VAR_INPUT
	{attribute 'OPC.UA.DA' := '1'}
	rAlarmHigh : REAL;
	{attribute 'OPC.UA.DA' := '1'}
	rAlarmLow : REAL;
	{attribute 'OPC.UA.DA' := '1'}
	rLimitHigh : REAL; // the upper limit of the desirable range (when the downward adjustment is activated)
	{attribute 'OPC.UA.DA' := '1'}
	rLimitLow : REAL; // lower limit of the desirable range (when the upward adjustment is activated)
	{attribute 'OPC.UA.DA' := '1'}
	nAdjustDelay : REAL; // min time in seconds between adjustments
	{attribute 'OPC.UA.DA' := '1'}
	nProcessValue : REAL; 
	{attribute 'OPC.UA.DA' := '1'}
	bEnabled : BOOL; 
	{attribute 'OPC.UA.DA' := '1'}
	rCurrentValue : REAL; 
	{attribute 'OPC.UA.DA' := '1'}
	sParameterName : STRING;
	{attribute 'OPC.UA.DA' := '1'}
	rSetpoint: REAL;
	{attribute 'OPC.UA.DA' := '1'}
	Mode:    E_CTRL_MODE;
END_VAR


VAR PERSISTENT

	n_ProcessValue: FLOAT;
	
	{attribute 'OPC.UA.DA' := '1'} 
	tPIDLoopTime: TIME := T#1M;	// how often the PID loop should be executed
	tResetMister: TIME := T#20M;	// reset the humidifiers every 20m so that the output doesn't get stuck high with mister ON timer expired causing mister to turn off
	
	// PID loop variables below
	nPID_Setpoint:			REAL; 
	nPID_SetpointBand:		REAL; // 
	nPID_ManSyncVal:		REAL;
	bPID_Sync: 				BOOL;
	nPID_Error:				REAL;
	nPID_ErrorPerc:			REAL;  
	nPID_Output: 			LREAL; 
	bPID_Hold: 				BOOL;
	ePID_Mode: 				E_CTRL_MODE;
	stPID_Parameters: 		ST_CTRL_PID_PARAMS;
	ePID_ErrorId: 			E_CTRL_ERRORCODES;
	bPID_Error: 			BOOL;
	bPID_ARWactive: 		BOOL;
	
	//stPIDParams values
	tPID_CtrlCycleTime: 		TIME := tPIDLoopTime;
	tPID_TaskCycleTime:			TIME := T#10MS;
	nPID_Kp:  					REAL := 1.0;
	nPID_Compensator:  			REAL := 1.0/1000.0;
	tPID_Tn: 					TIME := T#0S;
	tPID_Tv:					TIME := T#0S;
	tPID_Td:					TIME := T#200S; 
	nPID_OutMaxLimit: 			REAL := 300; 		// this is set in the cyclic routine, the error band moves with the setpoint
	nPID_OutMinLimit:			REAL := 0;
	bPID_PInTheFeedbackPath: 	BOOL := FALSE;
	bPID_DInTheFeedbackPath: 	BOOL := FALSE;
	bPID_ARWOnIPartOnly:		BOOL := FALSE;
	
	n_Output: LREAL := 0;
	
END_VAR

VAR
	bFirstRun: BOOL := TRUE;
	bResetTimer: BOOL := FALSE;
	
	eSMState: 	(WAIT, CALCULATE, TRIG_UP, TRIG_DOWN) := WAIT;

	{attribute 'OPC.UA.DA' := '0'} 
	fbTON_PIDLoop: TON := (PT := tPIDLoopTime, IN := FALSE);
	
	fbTON_OPCUATagReset: TON := (PT := T#1S, IN := FALSE);
	
	fbTON_ResetMister: TON := (PT := tResetMister, IN := FALSE);
	fbTON_ResetMisterCountdown: TON := (PT := T#1S, IN := FALSE);
	
	{attribute 'OPC.UA.DA' := '0'}
	PID: FB_CTRL_PID;
	
END_VAR


VAR_OUTPUT
	{attribute 'OPC.UA.DA' := '1'}
	bAdjustDownOutput 		AT %Q*: BOOL;
	{attribute 'OPC.UA.DA' := '1'}
	bAdjustUpOutput 		AT %Q*: BOOL;
	{attribute 'OPC.UA.DA' := '1'}
	bAlarmHigh : 			BOOL;
	{attribute 'OPC.UA.DA' := '1'}
	bAlarmLow : 			BOOL;
END_VAR


VAR
	fbTON_AdjustDown : 		TON;
	fbTON_AdjustUp : 		TON;
	{attribute 'OPC.UA.DA' := '1'}
	tAdjustUp : 			TIME;
	tAdjustDown : 			TIME;
	tAdjustUpCTRL : 			TIME; // these variables created to enable continuous misting - Ignition requires tAdjustUp/Down to be reset to 0 after each dose to enable plotting
	tAdjustDownCTRL : 			TIME;
	
END_VAR

IF bFirstRun THEN
	fbTON_PIDLoop(PT := tPIDLoopTime, IN := TRUE);
	fbTON_ResetMister(PT := tResetMister, IN := TRUE);
	bFirstRun := FALSE;
END_IF

//eState := eStateTarget;

IF (NOT bEnable) OR (eState = E_DeviceState.IDLE) THEN
	eState := E_DeviceState.IDLE;
	eStateTarget := E_DeviceState.IDLE;
	PID.eMode := E_CTRL_MODE.eCTRL_MODE_RESET;
END_IF

IF bEnable AND (eState = E_DeviceState.RUNNING) THEN
	PID.eMode := E_CTRL_MODE.eCTRL_MODE_ACTIVE;
END_IF 



// Execute timers
fbTON_PIDLoop(PT := tPIDLoopTime);
fbTON_OPCUATagReset();
fbTON_ResetMister();
fbTON_ResetMisterCountdown();

fbTON_AdjustUp();
fbTON_AdjustDown();

updatePIDParams();

nPID_Error 	:= nPID_Setpoint - nProcessValue; // calcuate error

nPID_Setpoint := (rLimitHigh + rLimitLow) / 2.0;
rSetpoint := (rLimitHigh + rLimitLow) / 2.0;

// nPID_Setpoint := 67;

rCurrentValue := nProcessValue;

IF fbTON_AdjustUp.Q THEN
	bAdjustUpOutput := FALSE;
	fbTON_AdjustUp.IN := FALSE;
END_IF

(*
IF fbTON_AdjustDown.Q THEN
	bAdjustDownOutput := FALSE;          // DEHUMIDIFER STAYS ON
	fbTON_AdjustDown.IN := FALSE;
END_IF
*)
bAdjustDownOutput := TRUE; // this code was added to keep the dehumidifier always on - remove this when we start controlling the fan

IF eState = E_DeviceState.RUNNING THEN
	//PID.eMode := E_CTRL_MODE.eCTRL_MODE_ACTIVE;
	PID( fSetpointValue := nPID_Setpoint, fActualValue := nProcessValue, stParams := stPID_Parameters);
END_IF


// IF control loop is ON and the loop timer has elapsed then enter the calculate / action state machine below
IF fbTON_PIDLoop.Q AND (eState = E_DeviceState.RUNNING) THEN
	fbTON_PIDLoop.IN := FALSE;
	eSMState := CALCULATE;		// This is the entry point to start PID calculations and dosing
END_IF

IF fbTON_OPCUATagReset.Q AND (eState = E_DeviceState.RUNNING) THEN
	tAdjustDown := T#0MS;
	tAdjustUp := T#0MS;
	fbTON_OPCUATagReset.IN := FALSE;
END_IF


CASE eSMState OF

	WAIT:
		// Do nothing and wait for timer to trigger
		fbTON_PIDLoop(IN := TRUE);
		
	
	CALCULATE:
	
		IF (eState = E_DeviceState.RUNNING) THEN 
			IF PID.fOut > 0 AND NOT fbTON_ResetMister.Q THEN
				tAdjustUp 	:= REAL_TO_TIME(PID.fOut) * 1000;
				tAdjustUpCTRL 	:= REAL_TO_TIME(PID.fOut) * 1000;
				tAdjustDown := T#0MS;
				eSMState 	:= TRIG_UP;
			ELSIF PID.fOut < 0 THEN
				tAdjustDown	:= REAL_TO_TIME(-PID.fOut) *1000;
				tAdjustDownCTRL	:= REAL_TO_TIME(-PID.fOut) *1000;
				tAdjustUp := T#0MS;
				eSMState 	:= TRIG_DOWN;
			END_IF
		END_IF
			
		fbTON_PIDLoop(IN := FALSE);
		fbTON_OPCUATagReset(IN := TRUE);  // set the OPCUA tag reset timer (Ignition requires these tags to be set to 0 to be visible on graph)
		
		//eSMState := WAIT;
		IF (eSMState <> TRIG_UP) AND (eSMState <> TRIG_DOWN) THEN
			eSMState := WAIT;
		END_IF
		
		
	TRIG_UP:
		fbTON_AdjustUp(PT := tAdjustUpCTRL, IN := TRUE);  // start the timer for the duration set at PID output
		bAdjustUpOutput := TRUE; // set output to high
		eSMState := WAIT; // go back to wait for the next timer trigger
		fbTON_PIDLoop(IN := TRUE);	// restart the PID loop timer

		
		
	TRIG_DOWN:
		fbTON_AdjustDown(PT := tAdjustDownCTRL, IN := TRUE); // start the timer for the duration set at PID output
		bAdjustDownOutput := TRUE; // set output to high
		eSMState := WAIT; // go back to wait for the next timer trigger
		fbTON_PIDLoop(IN := TRUE);			
		
		
END_CASE

IF fbTON_ResetMister.Q THEN

	fbTON_ResetMisterCountdown(IN := TRUE);
	fbTON_ResetMister(IN := FALSE);
END_IF

IF fbTON_ResetMisterCountdown.IN THEN
		bAdjustUpOutput := FALSE;	
END_IF
IF fbTON_ResetMisterCountdown.Q THEN
		fbTON_ResetMisterCountdown(IN := FALSE);
		fbTON_ResetMister(IN := TRUE);
END_IF

METHOD FB_init : BOOL
VAR_INPUT
	bInitRetains : BOOL; // if TRUE, the retain variables are initialized (warm start / cold start)
	bInCopyCode : BOOL;  // if TRUE, the instance afterwards gets moved into the copy code (online change)
	

	
END_VAR
END_METHOD

METHOD setParams : BOOL
VAR_INPUT
	(*
	NutrientMaxDoseRate: UINT;
	NutrientMinDoseRate: UINT;
	NutrientTimeBetweenDoses: TIME;
	PHMaxDoseRate: UINT;
	PHMinDoseRate: UINT;
	PHTimeBetweenDoses: TIME;


	// PID loop variables below
	*)
	Setpoint:		REAL; 
	(*
	NutrientSetpointBand:	REAL;
	NutrientManSyncVal:		REAL;
	NutrientSync: 			BOOL; 
	NutrientHold: 			BOOL;
	NutrientMode: 			E_CTRL_MODE;
	NutrientCtrlCycleTime: 	TIME;
	NutrientTaskCycleTime:	TIME;
	
	//stPIDParams values
	NutrientKp:  				REAL;
	NutrientTn: 				TIME; 
	NutrientTv:					TIME; 
	NutrientTd:					TIME; 
	NutrientOutMaxLimit: 		REAL;
	NutrientOutMinLimit:		REAL;
	NutrientPInTheFeedbackPath: BOOL;
	NutrientDInTheFeedbackPath: BOOL;
	NutrientARWOnIPartOnly:		BOOL;
	
	*)
	PHSetpoint:			REAL; 
	(*
	PHSetpointBand:		REAL;
	PHManSyncVal:		REAL;
	PHSync: 			BOOL;
	PHHold: 			BOOL;
	PHMode: 			E_CTRL_MODE;
	PHCtrlCycleTime: 		TIME;
	PHTaskCycleTime:		TIME;
	
	
	//stPIDParams values
	PHKp:  					REAL;
	PHTn: 					TIME;
	PHTv:					TIME;
	PHTd:					TIME; 
	PHOutMaxLimit: 			REAL; 		
	PHOutMinLimit:			REAL;
	PHPInTheFeedbackPath: 	BOOL;
	PHDInTheFeedbackPath:	BOOL;
	PHARWOnIPartOnly:		BOOL;
	*)
	
END_VAR
(*
nPIDNutrientMaxDoseRate := 				NutrientMaxDoseRate;
nPIDNutrientMinDoseRate := 				NutrientMinDoseRate;
tPIDNutrientTimeBetweenDoses := 		NutrientTimeBetweenDoses;

nPIDPHMaxDoseRate := 					PHMaxDoseRate;
nPIDPHMinDoseRate := 					PHMinDoseRate;
tPIDPHTimeBetweenDoses := 				PHTimeBetweenDoses;

*)
nPID_Setpoint := 						Setpoint;
(*
nPIDNutrientSetpointBand := 			NutrientSetpointBand;
nPIDNutrientManSyncVal := 				NutrientManSyncVal;
bPIDNutrientSync := 					NutrientSync;
bPIDNutrientHold := 					NutrientHold;
ePIDNutrientMode := 					NutrientMode;
tPIDNutrientCtrlCycleTime := 			NutrientCtrlCycleTime;
tPIDNutrientTaskCycleTime := 			NutrientTaskCycleTime;

nPIDNutrientKp := 						NutrientKp;
tPIDNutrientTn := 						NutrientTn;
tPIDNutrientTv := 						NutrientTv;
tPIDNutrientTd := 						NutrientTd;
nPIDNutrientOutMaxLimit := 				NutrientOutMaxLimit;
nPIDNutrientOutMinLimit := 				NutrientOutMinLimit;
bPIDNutrientPInTheFeedbackPath := 		NutrientPInTheFeedbackPath;
bPIDNutrientDInTheFeedbackPath := 		NutrientDInTheFeedbackPath;
bPIDNutrientARWactive := 				NutrientARWOnIPartOnly;
*)
END_METHOD

METHOD setState : BOOL
VAR_INPUT
	state : E_DeviceState;
END_VAR

eState := state;
END_METHOD

METHOD updatePIDParams : BOOL
VAR_INPUT
END_VAR


stPID_Parameters.tCtrlCycleTime := 		tPID_CtrlCycleTime;
stPID_Parameters.tTaskCycleTime := 		tPID_TaskCycleTime;
stPID_Parameters.fKp := 				nPID_Kp;
stPID_Parameters.tTn := 				tPID_Tn;
stPID_Parameters.tTv := 				tPID_Tv;
stPID_Parameters.tTd := 				tPID_Td;
stPID_Parameters.fOutMaxLimit := 		nPID_OutMaxLimit;
stPID_Parameters.fOutMinLimit := 		nPID_OutMinLimit;
stPID_Parameters.bPInTheFeedbackPath := bPID_PInTheFeedbackPath;
stPID_Parameters.bDInTheFeedbackPath := bPID_DInTheFeedbackPath;
stPID_Parameters.bARWOnIPartOnly := 	bPID_ARWOnIPartOnly;
END_METHOD

END_FUNCTION_BLOCK

// ---- POUs/04 Control Loops/Dosing Machine/FB_ControlLoop_PID_HVAC.TcPOU
FUNCTION_BLOCK FB_ControlLoop_PID_HVAC EXTENDS FB_BaseDevice


VAR_INPUT
	{attribute 'OPC.UA.DA' := '1'}
	rAlarmHigh : REAL;
	{attribute 'OPC.UA.DA' := '1'}
	rAlarmLow : REAL;
	{attribute 'OPC.UA.DA' := '1'}
	rLimitHigh : REAL; // the upper limit of the desirable range (when the downward adjustment is activated)
	{attribute 'OPC.UA.DA' := '1'}
	rLimitLow : REAL; // lower limit of the desirable range (when the upward adjustment is activated)
	{attribute 'OPC.UA.DA' := '1'}
	nAdjustDelay : REAL; // min time in seconds between adjustments
	{attribute 'OPC.UA.DA' := '1'}
	nProcessValue : REAL; 
	{attribute 'OPC.UA.DA' := '1'}
	bEnabled : BOOL; 
	{attribute 'OPC.UA.DA' := '1'}
	rCurrentValue : REAL; 
	{attribute 'OPC.UA.DA' := '1'}
	sParameterName : STRING;
	{attribute 'OPC.UA.DA' := '1'}
	rSetpoint: REAL;
	{attribute 'OPC.UA.DA' := '1'}
	Mode:    E_CTRL_MODE;
END_VAR


VAR PERSISTENT

	n_ProcessValue: FLOAT;
	
	{attribute 'OPC.UA.DA' := '1'} 
	tPIDLoopTime: TIME := T#1M;	// how often the PID loop should be executed
	
	// PID loop variables below
	nPID_Setpoint:			REAL; 
	nPID_SetpointBand:		REAL; // 
	nPID_ManSyncVal:		REAL;
	bPID_Sync: 				BOOL;
	nPID_Error:				REAL;
	nPID_ErrorPerc:			REAL;  
	nPID_Output: 			LREAL; 
	bPID_Hold: 				BOOL;
	ePID_Mode: 				E_CTRL_MODE;
	stPID_Parameters: 		ST_CTRL_PID_PARAMS;
	ePID_ErrorId: 			E_CTRL_ERRORCODES;
	bPID_Error: 			BOOL;
	bPID_ARWactive: 		BOOL;
	
	//stPIDParams values
	tPID_CtrlCycleTime: 		TIME := tPIDLoopTime;
	tPID_TaskCycleTime:			TIME := T#10MS;
	nPID_Kp:  					REAL := 1.0;
	nPID_Compensator:  			REAL := 1.0/1000.0;
	tPID_Tn: 					TIME := T#0S;
	tPID_Tv:					TIME := T#0S;
	tPID_Td:					TIME := T#200S; 
	nPID_OutMaxLimit: 			REAL := 300; 		// this is set in the cyclic routine, the error band moves with the setpoint
	nPID_OutMinLimit:			REAL := 0;
	bPID_PInTheFeedbackPath: 	BOOL := FALSE;
	bPID_DInTheFeedbackPath: 	BOOL := FALSE;
	bPID_ARWOnIPartOnly:		BOOL := FALSE;
	
	n_Output: LREAL := 0;
	
END_VAR

VAR
	bFirstRun: BOOL := TRUE;
	bResetTimer: BOOL := FALSE;
	
	eSMState: 	(WAIT, CALCULATE, TRIG_UP, TRIG_DOWN) := WAIT;

	{attribute 'OPC.UA.DA' := '0'} 
	fbTON_PIDLoop: TON := (PT := tPIDLoopTime, IN := FALSE);
	
	{attribute 'OPC.UA.DA' := '0'}
	PID: FB_CTRL_PID;
	
END_VAR


VAR_OUTPUT
	{attribute 'OPC.UA.DA' := '1'}
	bAdjustDownOutput 		AT %Q*: BOOL;
	{attribute 'OPC.UA.DA' := '1'}
	bAdjustUpOutput 		AT %Q*: BOOL;
	{attribute 'OPC.UA.DA' := '1'}
	bAlarmHigh : 			BOOL;
	{attribute 'OPC.UA.DA' := '1'}
	bAlarmLow : 			BOOL;
	{attribute 'OPC.UA.DA' := '1'}
	nControlValue:			REAL;
END_VAR


VAR
	fbTON_AdjustDown : 		TON;
	fbTON_AdjustUp : 		TON;
	tAdjustUp : 			TIME;
	tAdjustDown : 			TIME;
	
	{attribute 'OPC.UA.DA' := '1'}
	nControlValue: POINTER TO REAL;
	{attribute 'OPC.UA.DA' := '1'}
	nControlValueCopy: REAL;
	
END_VAR

IF bFirstRun THEN
	fbTON_PIDLoop(PT := tPIDLoopTime, IN := TRUE);
	bFirstRun := FALSE;
END_IF

//eState := eStateTarget;

IF (NOT bEnable) OR (eState = E_DeviceState.IDLE) THEN
	eState := E_DeviceState.IDLE;
	eStateTarget := E_DeviceState.IDLE;
	PID.eMode := E_CTRL_MODE.eCTRL_MODE_RESET;
END_IF

IF bEnable AND (eState = E_DeviceState.RUNNING) THEN
	PID.eMode := E_CTRL_MODE.eCTRL_MODE_ACTIVE;
END_IF 



// Execute timers
fbTON_PIDLoop(PT := tPIDLoopTime);
fbTON_AdjustUp();
fbTON_AdjustDown();

updatePIDParams();

nPID_Error 	:= nPID_Setpoint - nProcessValue; // calcuate error

nPID_Setpoint := (rLimitHigh + rLimitLow) / 2.0;

// nPID_Setpoint := 67;

rCurrentValue := nProcessValue;

(*
IF fbTON_AdjustDown.Q THEN
	bAdjustDownOutput := FALSE;
	fbTON_AdjustDown.IN := FALSE;
END_IF
*)

IF eState = E_DeviceState.RUNNING THEN
	PID( fSetpointValue := nPID_Setpoint, fActualValue := nProcessValue, stParams := stPID_Parameters);
END_IF


// IF control loop is ON and the loop timer has elapsed then enter the calculate / action state machine below
IF fbTON_PIDLoop.Q AND (eState = E_DeviceState.RUNNING) THEN
	fbTON_PIDLoop.IN := FALSE;
	eSMState := CALCULATE;		// This is the entry point to start PID calculations and dosing
END_IF



CASE eSMState OF

	WAIT:
		// Do nothing and wait for timer to trigger
		fbTON_PIDLoop(IN := TRUE);
	
	CALCULATE:
	
		nControlValue := nControlValue + PID.fOut;
		fbTON_PIDLoop(IN := FALSE);
		
		eSMState := WAIT;
		

		
	TRIG_UP:
		fbTON_AdjustUp(PT := tAdjustUp, IN := TRUE);  // start the timer for the duration set at PID output
		bAdjustUpOutput := TRUE; // set output to high
		eSMState := WAIT; // go back to wait for the next timer trigger
		fbTON_PIDLoop(IN := TRUE);	// restart the PID loop timer

		
		
	TRIG_DOWN:
		fbTON_AdjustDown(PT := tAdjustDown, IN := TRUE); // start the timer for the duration set at PID output
		bAdjustDownOutput := TRUE; // set output to high
		eSMState := WAIT; // go back to wait for the next timer trigger
		fbTON_PIDLoop(IN := TRUE);			
		
		
END_CASE

METHOD FB_init : BOOL
VAR_INPUT
	bInitRetains : BOOL; // if TRUE, the retain variables are initialized (warm start / cold start)
	bInCopyCode : BOOL;  // if TRUE, the instance afterwards gets moved into the copy code (online change)
	

	
END_VAR
END_METHOD

METHOD setParams : BOOL
VAR_INPUT
	(*
	NutrientMaxDoseRate: UINT;
	NutrientMinDoseRate: UINT;
	NutrientTimeBetweenDoses: TIME;
	PHMaxDoseRate: UINT;
	PHMinDoseRate: UINT;
	PHTimeBetweenDoses: TIME;


	// PID loop variables below
	*)
	Setpoint:		REAL; 
	(*
	NutrientSetpointBand:	REAL;
	NutrientManSyncVal:		REAL;
	NutrientSync: 			BOOL; 
	NutrientHold: 			BOOL;
	NutrientMode: 			E_CTRL_MODE;
	NutrientCtrlCycleTime: 	TIME;
	NutrientTaskCycleTime:	TIME;
	
	//stPIDParams values
	NutrientKp:  				REAL;
	NutrientTn: 				TIME; 
	NutrientTv:					TIME; 
	NutrientTd:					TIME; 
	NutrientOutMaxLimit: 		REAL;
	NutrientOutMinLimit:		REAL;
	NutrientPInTheFeedbackPath: BOOL;
	NutrientDInTheFeedbackPath: BOOL;
	NutrientARWOnIPartOnly:		BOOL;
	
	*)
	PHSetpoint:			REAL; 
	(*
	PHSetpointBand:		REAL;
	PHManSyncVal:		REAL;
	PHSync: 			BOOL;
	PHHold: 			BOOL;
	PHMode: 			E_CTRL_MODE;
	PHCtrlCycleTime: 		TIME;
	PHTaskCycleTime:		TIME;
	
	
	//stPIDParams values
	PHKp:  					REAL;
	PHTn: 					TIME;
	PHTv:					TIME;
	PHTd:					TIME; 
	PHOutMaxLimit: 			REAL; 		
	PHOutMinLimit:			REAL;
	PHPInTheFeedbackPath: 	BOOL;
	PHDInTheFeedbackPath:	BOOL;
	PHARWOnIPartOnly:		BOOL;
	*)
	
END_VAR
(*
nPIDNutrientMaxDoseRate := 				NutrientMaxDoseRate;
nPIDNutrientMinDoseRate := 				NutrientMinDoseRate;
tPIDNutrientTimeBetweenDoses := 		NutrientTimeBetweenDoses;

nPIDPHMaxDoseRate := 					PHMaxDoseRate;
nPIDPHMinDoseRate := 					PHMinDoseRate;
tPIDPHTimeBetweenDoses := 				PHTimeBetweenDoses;

*)
nPID_Setpoint := 						Setpoint;
(*
nPIDNutrientSetpointBand := 			NutrientSetpointBand;
nPIDNutrientManSyncVal := 				NutrientManSyncVal;
bPIDNutrientSync := 					NutrientSync;
bPIDNutrientHold := 					NutrientHold;
ePIDNutrientMode := 					NutrientMode;
tPIDNutrientCtrlCycleTime := 			NutrientCtrlCycleTime;
tPIDNutrientTaskCycleTime := 			NutrientTaskCycleTime;

nPIDNutrientKp := 						NutrientKp;
tPIDNutrientTn := 						NutrientTn;
tPIDNutrientTv := 						NutrientTv;
tPIDNutrientTd := 						NutrientTd;
nPIDNutrientOutMaxLimit := 				NutrientOutMaxLimit;
nPIDNutrientOutMinLimit := 				NutrientOutMinLimit;
bPIDNutrientPInTheFeedbackPath := 		NutrientPInTheFeedbackPath;
bPIDNutrientDInTheFeedbackPath := 		NutrientDInTheFeedbackPath;
bPIDNutrientARWactive := 				NutrientARWOnIPartOnly;
*)
END_METHOD

METHOD setState : BOOL
VAR_INPUT
	state : E_DeviceState;
END_VAR

eState := state;
END_METHOD

METHOD updatePIDParams : BOOL
VAR_INPUT
END_VAR
(*

stPID_Parameters.tCtrlCycleTime := 		tPID_CtrlCycleTime;
stPID_Parameters.tTaskCycleTime := 		tPID_TaskCycleTime;
stPID_Parameters.fKp := 				nPID_Kp;
stPID_Parameters.tTn := 				tPID_Tn;
stPID_Parameters.tTv := 				tPID_Tv;
stPID_Parameters.tTd := 				tPID_Td;
stPID_Parameters.fOutMaxLimit := 		nPID_OutMaxLimit;
stPID_Parameters.fOutMinLimit := 		nPID_OutMinLimit;
stPID_Parameters.bPInTheFeedbackPath := bPID_PInTheFeedbackPath;
stPID_Parameters.bDInTheFeedbackPath := bPID_DInTheFeedbackPath;
stPID_Parameters.bARWOnIPartOnly := 	bPID_ARWOnIPartOnly;

*)
END_METHOD

END_FUNCTION_BLOCK

// ---- POUs/04 Control Loops/Dosing Machine/FB_ControlLoop_TankLevel.TcPOU
(*
	Function Block which performs a level control using a DOL pump and a high level switch
*)
{attribute 'OPC.UA.DA.StructuredType' := '1'}
FUNCTION_BLOCK FB_ControlLoop_TankLevel EXTENDS FB_BaseDevice
VAR_IN_OUT
	fbValve: 	FB_Valve_ONOFF_woMonitoring;
	fbSensorH: 	FB_Sensor_SICKLevelSwitch_GRF18S;
END_VAR


VAR PERSISTENT
	tDebounce: TIME := T#1M; 
	tDebonce_Sensor: TIME := T#1.5S;
END_VAR

VAR
	bFirstRun: BOOL := TRUE;
	eSMState: (WAIT, FILLING, FULL, STOPPING);
	fbTON_Debouce: TON := (PT := tDebounce, IN := FALSE);
	
	
	fbTON_Debounce_Sensor: TON := (PT := tDebonce_Sensor, IN := FALSE);

END_VAR

IF bFirstRun THEN
	
	bFirstRun := FALSE;
END_IF

fbTON_Debounce_Sensor();
fbTON_Debouce();

IF GVL.bAutoUpdateDeviceState THEN
	eState := eStateTarget;	
END_IF

IF bEnable THEN
	fbValve.enable();
END_IF

IF eMode = E_DeviceMode.MANUAL THEN
	bEnable := TRUE;
END_IF

IF bEnable AND (eStateTarget = E_DeviceState.ON) AND eSMState <> FULL THEN
		eSMState := FILLING;
END_IF


IF (bEnable = FALSE OR eStateTarget = E_DeviceState.OFF) AND eSMState <> WAIT THEN
		eSMState := STOPPING;
END_IF


IF bEnable THEN
	CASE eSMState OF
		WAIT:
			// Do nothing
			eState := E_DeviceState.OFF;
		FILLING:
			fbTON_Debouce(IN := FALSE);
			eState := E_DeviceState.ON;
			fbValve.setCommand(StateTarget := E_DeviceState.OPEN);
			IF (fbSensorH.getValue() = 0) THEN
				eSMState := FULL;
				fbTON_Debounce_Sensor(IN := TRUE);
				IF fbTON_Debounce_Sensor.Q THEN
					eSMState := FULL;
					fbTON_Debounce_Sensor(IN := FALSE);
				END_IF
			END_IF
			
		FULL:
			fbTON_Debouce(PT := tDebounce, IN := TRUE);
			eState := E_DeviceState.ON;
			// Stop the pump
			fbValve.setCommand(StateTarget := E_DeviceState.CLOSED);
			IF (fbSensorH.getValue() = 1) AND (fbTON_Debouce.Q) THEN
				eSMState := FILLING;
			END_IF
			
		STOPPING:
			fbValve.setCommand(StateTarget := E_DeviceState.IDLE);
			eState := E_DeviceState.TURNING_OFF;
			eSMState := WAIT;	
	END_CASE
END_IF

METHOD setState : BOOL
VAR_INPUT
	state : E_DeviceState;
END_VAR

eState := state;
END_METHOD

END_FUNCTION_BLOCK

// ---- POUs/04 Control Loops/_ss/FB_ControlLoop_Dosing_1.TcPOU
FUNCTION_BLOCK FB_ControlLoop_Dosing_1 EXTENDS FB_BaseDevice

VAR
	bFirstRun: BOOL := TRUE;
	bResetTimer: BOOL := FALSE;
	
	nVolumeWater: REAL := 200.0; // Litres
	nHydrogenMoles: REAL;

		
	{attribute 'OPC.UA.DA' := '0'} 
	fbSensor_EC:	I_Sensor(SensorID := '', SensorDescr := '' , SensorType := E_SensorType.Analogue);
	{attribute 'OPC.UA.DA' := '0'} 
	fbSensor_DO:	I_Sensor(SensorID := '', SensorDescr := '' , SensorType := E_SensorType.Analogue);
	{attribute 'OPC.UA.DA' := '0'} 
	fbSensor_ORP:	I_Sensor(SensorID := '', SensorDescr := '' , SensorType := E_SensorType.Analogue);
	{attribute 'OPC.UA.DA' := '0'} 
	fbSensor_PH:	I_Sensor(SensorID := '', SensorDescr := '' , SensorType := E_SensorType.Analogue);
	{attribute 'OPC.UA.DA' := '0'} 
	fbSensor_TEMP:	I_Sensor(SensorID := '', SensorDescr := '' , SensorType := E_SensorType.Analogue);	

	{attribute 'OPC.UA.DA' := '0'} 
	fbDosingPump_phUp:  		I_PumpDosing;
	{attribute 'OPC.UA.DA' := '0'} 
	fbDosingPump_phDOwn:  		I_PumpDosing;
	{attribute 'OPC.UA.DA' := '0'} 
	fbDosingPump_Nutrient_A:  	I_PumpDosing;
	{attribute 'OPC.UA.DA' := '0'} 
	fbDosingPump_Nutrient_B:  	I_PumpDosing;
	{attribute 'OPC.UA.DA' := '0'} 
	fbDosingPump_Nutrient_C:  	I_PumpDosing;
	{attribute 'OPC.UA.DA' := '0'} 
	eSMState: 					(INIT, WAIT_TRIG, WAIT, NUTRIENT_ONLY, NUTRIENT_AND_PH) := INIT;
	{attribute 'OPC.UA.DA' := '0'} 
	eCurrentNutrient: 			(NUTRIENT_A,NUTRIENT_B,NUTRIENT_C, PH) := NUTRIENT_C;
	
	
	bDoseRequestSent:		BOOL := FALSE;
	bDoseRequestComplete: 	BOOL := FALSE;
	
	nPIDNutrientMaxDoseRate: UINT;
	nPIDNutrientMinDoseRate: UINT;
	tPIDNutrientTimeBetweenDoses: TIME;
	nPIDPHMaxDoseRate: UINT;
	nPIDPHMinDoseRate: UINT;
	tPIDPHTimeBetweenDoses: TIME;
	
	{attribute 'OPC.UA.DA' := '0'} 
	fbTON_PIDLoop: TON := (PT := tPIDLoopTime, IN := FALSE);
	{attribute 'OPC.UA.DA' := '1'} 
	tPIDLoopTime: TIME := T#10S;			//5 second PID calculation


	// PID loop variables below
	nPIDNutrientSetpoint:		REAL; 
	nPIDNutrientSetpointBand:	REAL; // %
	nPIDNutrientManSyncVal:		REAL;
	bPIDNutrientSync: 			BOOL;
	nPIDNutrientError:			REAL;
	nPIDNutrientErrorPerc:		REAL;  // this is used to check if we are at 75%
	nPIDNutrientOutput: 		LREAL; 
	bPIDNutrientHold: 			BOOL;
	ePIDNutrientMode: 			E_CTRL_MODE;
	stPIDNutrientParameters: 	ST_CTRL_PID_PARAMS;
	ePIDNutrientErrorId: 		E_CTRL_ERRORCODES;
	bPIDNutrientError: 			BOOL;
	bPIDNutrientARWactive: 		BOOL;
	
	//stPIDParams values
	tPIDNutrientCtrlCycleTime: 		TIME;
	tPIDNutrientTaskCycleTime:		TIME;
	nPIDNutrientKp:  				REAL;
	tPIDNutrientTn: 				TIME; 
	tPIDNutrientTv:					TIME; 
	tPIDNutrientTd:					TIME; 
	nPIDNutrientOutMaxLimit: 		REAL; 		// this is set in the cyclic routine, the error band moves with the setpoint
	nPIDNutrientOutMinLimit:		REAL;
	bPIDNutrientPInTheFeedbackPath: BOOL;
	bPIDNutrientDInTheFeedbackPath: BOOL;
	bPIDNutrientARWOnIPartOnly:		BOOL;
	
	{attribute 'OPC.UA.DA' := '0'}
	PID_Nutrient: FB_CTRL_PID;
	
	// Inputs
	nPIDPHSetpoint:			FLOAT; 					// Setpoint of the controlled variable (units pH)
	nPIDPHSetpoint_HydrogenMoles:	FLOAT;			// Setpoint of the controlled variable (H+ moles)
	nPIDPHSetpointBand:		REAL;					// 
	nPIDPHManSyncVal:		REAL;					// 	Input, to whose value it is possible to set the internal state of the PID-element.
	bPIDPHSync: 			BOOL;					//  A rising edge at this input sets the PID-element to the value "fManSyncValue".
	nPIDPHError:			REAL;					//  This is abs(actual - setpoint)

	bPIDPHHold: 			BOOL;					// 	A TRUE at this input will hold the internal state (and therefore also the output) constant at its current value, independently of the control deviation.			
	ePIDPHMode: 			E_CTRL_MODE;			//  Input that specifies the operation mode of the function block.
	
	
	// Outputs 
	nPIDPHOutput: 			LREAL;					// Output of the PID element
	ePIDPHErrorId: 			E_CTRL_ERRORCODES;		// Supplies the error number when the output bError is set.
	bPIDPHError: 			BOOL;					// Becomes TRUE, as soon as an error occurs.
	bPIDPHARWactive: 		BOOL;					// A TRUE at this output indicates that the PID-element is being restricted.
	
	// Inputs & Outputs (VAR IN OUT)
	stPIDPHParameters: 		ST_CTRL_PID_PARAMS;		// Parameter structure of the PID element
	
	//stPIDParams values
	tPIDPHCtrlCycleTime: 		TIME := T#10S;	// Cycle time with which the control loop is processed. This must be greater than or equal to the TaskCycleTime. The function block uses this input value to calculate internally whether the state and the output values have to be updated in the current cycle.
	tPIDPHTaskCycleTime:		TIME := T#10S;	// Cycle TIME with which the FUNCTION block is called. IF the FUNCTION block is called in every cycle THIS corresponds TO the task cycle TIME OF the calling task
	nPIDPHKp:  					FLOAT;  		// Controller amplification / controller coefficient
	tPIDPHTn: 					TIME;  			// Integral action time; if this is parameterized to T#0s, the I component is deactivated.
	tPIDPHTv:					TIME := T#0S;  	// Derivative action time; if this is parameterized to T#0s, the D component is deactivated.
	tPIDPHTd:					TIME; 			// Damping time
	nPIDPHOutMaxLimit: 			REAL; 			// Upper limit at which integration is halted and to which the output is limited (ARW measure). Reaching this limit is indicated by a TRUE at the bARWActive output.
	nPIDPHOutMinLimit:			REAL;			// 	Lower LIMIT AT which integration is halted AND TO which the output is limited (ARW measure). Reaching THIS LIMIT is indicated BY a TRUE AT the bARWActive output
	bPIDPHPInTheFeedbackPath: 	BOOL := FALSE;	// Input value of the internal P-element can be selected with this input (see functional diagram). Standard setting: FALSE
	bPIDPHDInTheFeedbackPath:	BOOL := FALSE;	//  Input value of the internal D-element can be selected with this input (see functional diagram). Standard setting: FALSE
	bPIDPHARWOnIPartOnly:		BOOL;			// 	If this parameter is FALSE (the standard setting), the integration of the I-component is halted if the complete controller output reaches the upper or lower limit. If it is TRUE, the integration is halted if the I-component (the output of the integrator) reaches some limit. (Cf. functional diagram.)
	
	{attribute 'OPC.UA.DA' := '0'}
	PID_PH: FB_CTRL_PID;
	
END_VAR

IF bFirstRun THEN
	fbTON_PIDLoop(PT := tPIDLoopTime, IN := TRUE);
END_IF

fbTON_PIDLoop();

CASE eState OF
	
	INIT:
		updatePIDParams();
		eSMState := WAIT_TRIG;

	WAIT_TRIG:
	
		fbTON_PIDLoop(IN:= TRUE, PT := tPIDLoopTime); // this controls the PID control loop cycle time
		nPIDNutrientError := nPIDNutrientSetpoint - fbSensor_EC.getValue(); //fbSM.getEC();
		
		IF nPIDNutrientSetpoint > 0 THEN
			nPIDNutrientErrorPerc:=	1 - (ABS(nPIDNutrientError)/nPIDNutrientSetpoint); // this is used to decide if we opt for nutrient only dosing or nutrient and PH
		ELSE
			nPIDNutrientErrorPerc:=	0.9;
		END_IF
		nPIDPHError:= nPIDPHSetpoint - fbSensor_PH.getValue();
		
		IF fbTON_PIDLoop.Q THEN
			eSMState := WAIT;
			fbTON_PIDLoop.IN := FALSE;	
		END_IF
		
	
	WAIT:

		IF nPIDNutrientErrorPerc < 0.75 THEN    // only bring in pH when EC is 75% percent of setpoint
			eSMState := NUTRIENT_ONLY;
		ELSE
			eSMState := NUTRIENT_AND_PH;
		END_IF

		
		
	NUTRIENT_ONLY:
		
		nPIDNutrientOutMaxLimit := ( 1 + nPIDNutrientSetpointBand) * nPIDNutrientSetpoint;
		nPIDNutrientOutMinLimit := ( 1 - nPIDNutrientSetpointBand) * nPIDNutrientSetpoint;
		stPIDNutrientParameters.fOutMaxLimit := nPIDNutrientOutMaxLimit;
		stPIDNutrientParameters.fOutMinLimit := nPIDNutrientOutMinLimit;
	
		PID_Nutrient(	fSetpointValue		:= nPIDNutrientSetpoint,
						fActualValue		:= fbSensor_EC.getValue(),
						fManSyncValue		:= nPIDNutrientManSyncVal,
						bSync				:= bPIDNutrientSync,
						eMode				:= ePIDNutrientMode,
						bHold				:= bPIDNutrientHold,
						stParams			:= stPIDNutrientParameters,
						fOut				=> nPIDNutrientOutput,
						bARWactive			=> bPIDNutrientARWactive,
						eErrorId			=> ePIDNutrientErrorId,
						bError				=> bPIDNutrientError );
		
						
		// Handle the case where we have transitioned from dosing Nutrient+PH to Nutrient only (reset nutrient order)
		IF eCurrentNutrient = PH THEN
			eCurrentNutrient := NUTRIENT_A;
		END_IF				
		
		
		CASE eCurrentNutrient OF 
			
			NUTRIENT_A:
				IF nPIDNutrientError > 0 AND bDoseRequestSent = FALSE THEN
					fbDosingPump_Nutrient_A.executeDose(DoseQtyMls := LREAL_TO_UINT(nPIDNutrientOutput), DoseRateMlph := 40, RequestComplete := ADR(bDoseRequestComplete), RequestAccepted => bDoseRequestSent); // change arbitrary 40 lph to a variable based on dose amount

				ELSIF bDoseRequestSent = TRUE AND bDoseRequestComplete = TRUE THEN
					eCurrentNutrient	:= NUTRIENT_B;
					bDoseRequestSent 	:= FALSE;
					bDoseRequestComplete:= FALSE;
				ELSIF  nPIDNutrientError < 0 THEN // EC is overdosed
					eCurrentNutrient	:= PH;
				END_IF
				
			NUTRIENT_B:
			
				IF nPIDNutrientError > 0 AND bDoseRequestSent = FALSE THEN
					fbDosingPump_Nutrient_B.executeDose(DoseQtyMls := LREAL_TO_UINT(nPIDNutrientOutput), DoseRateMlph := 40, RequestComplete := ADR(bDoseRequestComplete), RequestAccepted => bDoseRequestSent); // change arbitrary 40 lph to a variable based on dose amount 
					
				ELSIF bDoseRequestSent = TRUE AND bDoseRequestComplete = TRUE THEN
					eCurrentNutrient	:= NUTRIENT_C;
					bDoseRequestSent 	:= FALSE;
					bDoseRequestComplete:= FALSE;
				ELSIF  nPIDNutrientError < 0 THEN 
					eCurrentNutrient	:= PH;
				END_IF

				
			NUTRIENT_C:
			
				IF nPIDNutrientError > 0 AND bDoseRequestSent = FALSE THEN
						fbDosingPump_Nutrient_C.executeDose(DoseQtyMls := LREAL_TO_UINT(nPIDNutrientOutput), DoseRateMlph := 40, RequestComplete := ADR(bDoseRequestComplete), RequestAccepted => bDoseRequestSent); // change arbitrary 40 lph to a variable based on dose amount 
						
				ELSIF bDoseRequestSent = TRUE AND bDoseRequestComplete = TRUE THEN
						eCurrentNutrient	:= PH;
						bDoseRequestSent 	:= FALSE;
						bDoseRequestComplete:= FALSE;
				ELSIF  nPIDNutrientError < 0 THEN 
					eCurrentNutrient	:= NUTRIENT_A;
				END_IF
		END_CASE

		
		
	NUTRIENT_AND_PH:
	
		PID_Nutrient(	fSetpointValue		:= nPIDNutrientSetpoint,
						fActualValue		:= fbSensor_EC.getValue(),
						fManSyncValue		:= nPIDNutrientManSyncVal,
						bSync				:= bPIDNutrientSync,
						eMode				:= ePIDNutrientMode,
						bHold				:= bPIDNutrientHold,
						stParams			:= stPIDNutrientParameters,
						fOut				=> nPIDNutrientOutput,
						bARWactive			=> bPIDNutrientARWactive,
						eErrorId			=> ePIDNutrientErrorId,
						bError				=> bPIDNutrientError );
						
		PID_PH(			fSetpointValue		:= nPIDPHSetpoint_HydrogenMoles,
						fActualValue		:= nHydrogenMoles,
						fManSyncValue		:= nPIDPHManSyncVal,
						bSync				:= bPIDPHSync,
						eMode				:= ePIDPHMode,
						bHold				:= bPIDPHHold,
						stParams			:= stPIDPHParameters,
						fOut				=> nPIDPHOutput,
						bARWactive			=> bPIDPHARWactive,
						eErrorId			=> ePIDPHErrorId,
						bError				=> bPIDPHError );
						
						
		
		
		// Commdand pump to dose desired amount from PID loops - rotate A,B,C and pH pumps
		CASE eCurrentNutrient OF 
			
			NUTRIENT_A:
				IF nPIDNutrientError > 0 AND bDoseRequestSent = FALSE THEN
					fbDosingPump_Nutrient_A.executeDose(DoseQtyMls := LREAL_TO_UINT(nPIDNutrientOutput), DoseRateMlph := 40, RequestComplete := ADR(bDoseRequestComplete), RequestAccepted => bDoseRequestSent); // change arbitrary 40 lph to a variable based on dose amount 
					
				ELSIF bDoseRequestSent = TRUE AND bDoseRequestComplete = TRUE THEN
					eCurrentNutrient	:= NUTRIENT_B;
					bDoseRequestSent 	:= FALSE;
					bDoseRequestComplete:= FALSE;
				ELSIF  nPIDNutrientError < 0 THEN // EC is overdosed
					eCurrentNutrient	:= PH;
				END_IF
				
			NUTRIENT_B:
			
				IF nPIDNutrientError > 0 AND bDoseRequestSent = FALSE THEN
					fbDosingPump_Nutrient_B.executeDose(DoseQtyMls := LREAL_TO_UINT(nPIDNutrientOutput), DoseRateMlph := 40, RequestComplete := ADR(bDoseRequestComplete), RequestAccepted => bDoseRequestSent); // change arbitrary 40 lph to a variable based on dose amount 
					
				ELSIF bDoseRequestSent = TRUE AND bDoseRequestComplete = TRUE THEN
					eCurrentNutrient	:= NUTRIENT_C;
					bDoseRequestSent 	:= FALSE;
					bDoseRequestComplete:= FALSE;
				ELSIF  nPIDNutrientError < 0 THEN 
					eCurrentNutrient	:= PH;
				END_IF

				
			NUTRIENT_C:
			
				IF nPIDNutrientError > 0 AND bDoseRequestSent = FALSE THEN
					fbDosingPump_Nutrient_C.executeDose(DoseQtyMls := LREAL_TO_UINT(nPIDNutrientOutput), DoseRateMlph := 40, RequestComplete := ADR(bDoseRequestComplete), RequestAccepted => bDoseRequestSent); // change arbitrary 40 lph to a variable based on dose amount 
						
				ELSIF bDoseRequestSent = TRUE AND bDoseRequestComplete = TRUE THEN
						eCurrentNutrient	:= PH;
						bDoseRequestSent 	:= FALSE;
						bDoseRequestComplete:= FALSE;
				ELSIF  nPIDNutrientError < 0 THEN 
					eCurrentNutrient	:= PH;
				END_IF

			PH:
				IF nPIDPHError > 0 AND bDoseRequestSent = FALSE THEN
					fbDosingPump_phUp.executeDose(DoseQtyMls := LREAL_TO_UINT(nPIDPHOutput), DoseRateMlph := 40, RequestComplete := ADR(bDoseRequestComplete), RequestAccepted => bDoseRequestSent); // change arbitrary 40 lph to a variable based on dose amount
				ELSIF nPIDPHError < 0 AND bDoseRequestSent = FALSE THEN
					fbDosingPump_phDown.executeDose(DoseQtyMls := LREAL_TO_UINT(nPIDPHOutput), DoseRateMlph := 40, RequestComplete := ADR(bDoseRequestComplete), RequestAccepted => bDoseRequestSent); // change arbitrary 40 lph to a variable based on dose amount
				ELSIF bDoseRequestSent = TRUE AND bDoseRequestComplete = TRUE THEN
					eCurrentNutrient	:= NUTRIENT_A;
					bDoseRequestSent 	:= FALSE;
					bDoseRequestComplete:= FALSE;
				END_IF
		END_CASE
						
		eSMState := WAIT_TRIG;
						
		
END_CASE

METHOD calcMoles : BOOL
VAR_INPUT
END_VAR
nHydrogenMoles := EXPT(10, fbSensor_PH.getValue());
nPIDPHSetpoint_HydrogenMoles := EXPT(10, nPIDPHSetpoint);
END_METHOD

METHOD FB_init : BOOL
VAR_INPUT
	bInitRetains : BOOL; // if TRUE, the retain variables are initialized (warm start / cold start)
	bInCopyCode : BOOL;  // if TRUE, the instance afterwards gets moved into the copy code (online change)
	
	DosingPump_phUp:  			I_PumpDosing;
	DosingPump_phDOwn:  		I_PumpDosing;
	DosingPump_Nutrient_A:  	I_PumpDosing;
	DosingPump_Nutrient_B:  	I_PumpDosing;
	DosingPump_Nutrient_C:  	I_PumpDosing;
	
	Sensor_EC:				I_Sensor(SensorID := '', SensorDescr := '' , SensorType := E_SensorType.Analogue);
	Sensor_DO:				I_Sensor(SensorID := '', SensorDescr := '' , SensorType := E_SensorType.Analogue);
	Sensor_ORP:				I_Sensor(SensorID := '', SensorDescr := '' , SensorType := E_SensorType.Analogue);
	Sensor_PH:				I_Sensor(SensorID := '', SensorDescr := '' , SensorType := E_SensorType.Analogue);
	Sensor_TEMP:			I_Sensor(SensorID := '', SensorDescr := '' , SensorType := E_SensorType.Analogue);
	
END_VAR
fbDosingPump_phUp 		:= DosingPump_phUp;
fbDosingPump_phDOwn 	:= DosingPump_phDOwn;
fbDosingPump_Nutrient_A := DosingPump_Nutrient_A;
fbDosingPump_Nutrient_B := DosingPump_Nutrient_B;
fbDosingPump_Nutrient_C := DosingPump_Nutrient_C;

fbSensor_EC := Sensor_EC;
fbSensor_DO := Sensor_DO;
fbSensor_ORP := Sensor_ORP;
fbSensor_PH := Sensor_PH;
fbSensor_TEMP := Sensor_TEMP;
END_METHOD

// This method is used by the Scan OPC inputs method
METHOD setParams : BOOL
VAR_INPUT
	
	NutrientMaxDoseRate: UINT;
	NutrientMinDoseRate: UINT;
	NutrientTimeBetweenDoses: TIME;
	PHMaxDoseRate: UINT;
	PHMinDoseRate: UINT;
	PHTimeBetweenDoses: TIME;


	// PID loop variables below
	NutrientSetpoint:		REAL; 
	NutrientSetpointBand:	REAL;
	NutrientManSyncVal:		REAL;
	NutrientSync: 			BOOL; 
	NutrientHold: 			BOOL;
	NutrientMode: 			E_CTRL_MODE;
	NutrientCtrlCycleTime: 	TIME;
	NutrientTaskCycleTime:	TIME;
	
	//stPIDParams values
	NutrientKp:  				REAL;
	NutrientTn: 				TIME; 
	NutrientTv:					TIME; 
	NutrientTd:					TIME; 
	NutrientOutMaxLimit: 		REAL;
	NutrientOutMinLimit:		REAL;
	NutrientPInTheFeedbackPath: BOOL;
	NutrientDInTheFeedbackPath: BOOL;
	NutrientARWOnIPartOnly:		BOOL;
	
	
	PHSetpoint:			REAL; 
	PHSetpointBand:		REAL;
	PHManSyncVal:		REAL;
	PHSync: 			BOOL;
	PHHold: 			BOOL;
	PHMode: 			E_CTRL_MODE;
	PHCtrlCycleTime: 		TIME;
	PHTaskCycleTime:		TIME;
	
	
	//stPIDParams values
	PHKp:  					REAL;
	PHTn: 					TIME;
	PHTv:					TIME;
	PHTd:					TIME; 
	PHOutMaxLimit: 			REAL; 		
	PHOutMinLimit:			REAL;
	PHPInTheFeedbackPath: 	BOOL;
	PHDInTheFeedbackPath:	BOOL;
	PHARWOnIPartOnly:		BOOL;

	
END_VAR
nPIDNutrientMaxDoseRate := 				NutrientMaxDoseRate;
nPIDNutrientMinDoseRate := 				NutrientMinDoseRate;
tPIDNutrientTimeBetweenDoses := 		NutrientTimeBetweenDoses;

nPIDPHMaxDoseRate := 					PHMaxDoseRate;
nPIDPHMinDoseRate := 					PHMinDoseRate;
tPIDPHTimeBetweenDoses := 				PHTimeBetweenDoses;


nPIDNutrientSetpoint := 				NutrientSetpoint;
nPIDNutrientSetpointBand := 			NutrientSetpointBand;
nPIDNutrientManSyncVal := 				NutrientManSyncVal;
bPIDNutrientSync := 					NutrientSync;
bPIDNutrientHold := 					NutrientHold;
ePIDNutrientMode := 					NutrientMode;
tPIDNutrientCtrlCycleTime := 			NutrientCtrlCycleTime;
tPIDNutrientTaskCycleTime := 			NutrientTaskCycleTime;

nPIDNutrientKp := 						NutrientKp;
tPIDNutrientTn := 						NutrientTn;
tPIDNutrientTv := 						NutrientTv;
tPIDNutrientTd := 						NutrientTd;
nPIDNutrientOutMaxLimit := 				NutrientOutMaxLimit;
nPIDNutrientOutMinLimit := 				NutrientOutMinLimit;
bPIDNutrientPInTheFeedbackPath := 		NutrientPInTheFeedbackPath;
bPIDNutrientDInTheFeedbackPath := 		NutrientDInTheFeedbackPath;
bPIDNutrientARWactive := 				NutrientARWOnIPartOnly;

nPIDPHSetpoint := 						PHSetpoint;
nPIDPHSetpointBand := 					PHSetpointBand;
nPIDPHManSyncVal := 					PHManSyncVal;
bPIDPHSync := 							PHSync;
bPIDPHHold := 							PHHold;
ePIDPHMode := 							PHMode;
tPIDPHCtrlCycleTime := 					PHCtrlCycleTime;
tPIDPHTaskCycleTime := 					PHTaskCycleTime;

nPIDPHKp := 							PHKp;
tPIDPHTn := 							PHTn;
tPIDPHTv := 							PHTv;
tPIDPHTd := 							PHTd;
nPIDPHOutMaxLimit := 					PHOutMaxLimit;
nPIDPHOutMinLimit := 					PHOutMinLimit;
bPIDPHPInTheFeedbackPath := 			PHPInTheFeedbackPath;
bPIDPHDInTheFeedbackPath := 			PHDInTheFeedbackPath;
bPIDPHARWactive := 						PHARWOnIPartOnly;
END_METHOD

METHOD updatePIDParams : BOOL
VAR_INPUT
END_VAR
stPIDNutrientParameters.tCtrlCycleTime := tPIDNutrientCtrlCycleTime;
stPIDNutrientParameters.tTaskCycleTime := tPIDNutrientTaskCycleTime;
stPIDNutrientParameters.fKp := nPIDNutrientKp;
stPIDNutrientParameters.tTn := tPIDNutrientTn;
stPIDNutrientParameters.tTv := tPIDNutrientTv;
stPIDNutrientParameters.tTd := tPIDNutrientTd;
stPIDNutrientParameters.fOutMaxLimit := nPIDNutrientOutMaxLimit;
stPIDNutrientParameters.fOutMinLimit := nPIDNutrientOutMinLimit;
stPIDNutrientParameters.bPInTheFeedbackPath := bPIDNutrientPInTheFeedbackPath;
stPIDNutrientParameters.bDInTheFeedbackPath := bPIDNutrientDInTheFeedbackPath;
stPIDNutrientParameters.bARWOnIPartOnly := bPIDNutrientARWOnIPartOnly;

stPIDPHParameters.tCtrlCycleTime := tPIDPHCtrlCycleTime;
stPIDPHParameters.tTaskCycleTime := tPIDPHTaskCycleTime;
stPIDPHParameters.fKp := nPIDPHKp;
stPIDPHParameters.tTn := tPIDPHTn;
stPIDPHParameters.tTv := tPIDPHTv;
stPIDPHParameters.tTd := tPIDPHTd;
stPIDPHParameters.fOutMaxLimit := nPIDPHOutMaxLimit;
stPIDPHParameters.fOutMinLimit := nPIDPHOutMinLimit;
stPIDPHParameters.bPInTheFeedbackPath := bPIDPHPInTheFeedbackPath;
stPIDPHParameters.bDInTheFeedbackPath := bPIDPHDInTheFeedbackPath;
stPIDPHParameters.bARWOnIPartOnly := bPIDPHARWOnIPartOnly;
END_METHOD

END_FUNCTION_BLOCK

// ---- POUs/05 Sequences/Dosing Machine/FB_SequenceDM_Calibrate.TcPOU
FUNCTION_BLOCK FB_SequenceDM_Calibrate EXTENDS FB_SequenceBase

VAR
	bUseMainPump_A: BOOL := TRUE;  // this boolean is used to keep track of which of the two redudant pumps we should use
END_VAR

VAR_IN_OUT
	devices: ST_DMComponents;
END_VAR

METHOD FB_init : BOOL
VAR_INPUT
	bInitRetains : BOOL; // if TRUE, the retain variables are initialized (warm start / cold start)
	bInCopyCode : BOOL;  // if TRUE, the instance afterwards gets moved into the copy code (online change)
END_VAR
(*
		Here we set the order of things to command, what the commands should be, and also how much time to allow during and between steps
		Every component listed below becomes 'Enabled' at each step
*)
sSequenceName := 'DM Calibrate SEQ';
sSequenceName := 'Dosing Machine Calibrate sequence';

(*
Step9.Component := 
Step9.Command :=
Step9.StepMinDuration :=
Step9.DelayUntilNextStep :=
 
Step10.Component :=
Step10.Command :=
Step10.StepMinDuration :=
Step10.DelayUntilNextStep :=
 
Step11.Component :=
Step11.Command :=
Step11.StepMinDuration :=
Step11.DelayUntilNextStep :=
 
Step12.Component :=
Step12.Command :=
Step12.StepMinDuration :=
Step12.DelayUntilNextStep :=
 
Step13.Component :=
Step13.Command :=
Step13.StepMinDuration :=
Step13.DelayUntilNextStep :=
 
Step14.Component :=
Step14.Command :=
Step14.StepMinDuration :=
Step14.DelayUntilNextStep :=
 
Step15.Component :=
Step15.Command :=
Step15.StepMinDuration :=
Step15.DelayUntilNextStep :=
 
Step16.Component :=
Step16.Command :=
Step16.StepMinDuration :=
Step16.DelayUntilNextStep :=
 
Step17.Component :=
Step17.Command :=
Step17.StepMinDuration :=
Step17.DelayUntilNextStep :=
 
Step18.Component :=
Step18.Command :=
Step18.StepMinDuration :=
Step18.DelayUntilNextStep :=
 
Step19.Component :=
Step19.Command :=
Step19.StepMinDuration :=
Step19.DelayUntilNextStep :=
 
Step20.Component :=
Step20.Command :=
Step20.StepMinDuration :=
Step20.DelayUntilNextStep :=
 
Step21.Component :=
Step21.Command :=
Step21.StepMinDuration :=
Step21.DelayUntilNextStep :=
 
Step22.Component :=
Step22.Command :=
Step22.StepMinDuration :=
Step22.DelayUntilNextStep :=
 
Step23.Component :=
Step23.Command :=
Step23.StepMinDuration :=
Step23.DelayUntilNextStep :=
 
Step24.Component :=
Step24.Command :=
Step24.StepMinDuration :=
Step24.DelayUntilNextStep :=
 
Step25.Component :=
Step25.Command :=
Step25.StepMinDuration :=
Step25.DelayUntilNextStep :=
 
Step26.Component :=
Step26.Command :=
Step26.StepMinDuration :=
Step26.DelayUntilNextStep :=
 
Step27.Component :=
Step27.Command :=
Step27.StepMinDuration :=
Step27.DelayUntilNextStep :=
 
Step28.Component :=
Step28.Command :=
Step28.StepMinDuration :=
Step28.DelayUntilNextStep :=
 
Step29.Component :=
Step29.Command :=
Step29.StepMinDuration :=
Step29.DelayUntilNextStep :=
 
Step30.Component :=
Step30.Command :=
Step30.StepMinDuration :=
Step30.DelayUntilNextStep :=
 
Step31.Component :=
Step31.Command :=
Step31.StepMinDuration :=
Step31.DelayUntilNextStep :=
 
Step32.Component :=
Step32.Command :=
Step32.StepMinDuration :=
Step32.DelayUntilNextStep :=
 
Step33.Component :=
Step33.Command :=
Step33.StepMinDuration :=
Step33.DelayUntilNextStep :=
 
Step34.Component :=
Step34.Command :=
Step34.StepMinDuration :=
Step34.DelayUntilNextStep :=
 
Step35.Component :=
Step35.Command :=
Step35.StepMinDuration :=
Step35.DelayUntilNextStep :=
 
Step36.Component :=
Step36.Command :=
Step36.StepMinDuration :=
Step36.DelayUntilNextStep :=
 
Step37.Component :=
Step37.Command :=
Step37.StepMinDuration :=
Step37.DelayUntilNextStep :=
 
Step38.Component :=
Step38.Command :=
Step38.StepMinDuration :=
Step38.DelayUntilNextStep :=
 
Step39.Component :=
Step39.Command :=
Step39.StepMinDuration :=
Step39.DelayUntilNextStep :=

*)
END_METHOD

METHOD populateSteps : ST_SequenceStep
VAR_INPUT

END_VAR
(*
		Here we set the order of things to command, what the commands should be, and also how much time to allow during and between steps
		Every component listed below becomes 'Enabled' at each step
*)
sSequenceName := 'DM Calibrate SEQ';
sSequenceName := 'Dosing Machine Calibrate sequence';

Step1.Device := ADR(devices.fbValve_DosingSupply^);
//Step1.Component := devices.fbControlLoop_Dosing;			
Step1.Command := E_DeviceState.IDLE;
Step1.StepMinDuration := T#0S;
Step1.DelayUntilNextStep := T#5S; // allow sufficient time to clear the dosing line
aSequenceSteps[1] := Step1;
 
Step2.Device := ADR(devices.fbStrainer^);
Step2.Command := E_DeviceState.RUNNING;
Step2.StepMinDuration := T#0S;
Step2.DelayUntilNextStep := T#0S;
aSequenceSteps[2] := Step2;
 
Step3.Device := ADR(devices.fbUnit_UltraSonCleaner^);
Step3.Command := E_DeviceState.ON;
Step3.StepMinDuration := T#0S;
Step3.DelayUntilNextStep := T#0S;
aSequenceSteps[3] := Step3;
 
Step4.Device := ADR(Devices.fbUVFilter1^);
Step4.Command := E_DeviceState.ON;
Step4.StepMinDuration := T#0S;
Step4.DelayUntilNextStep := T#0S;
aSequenceSteps[4] := Step4;


Step5.Device := ADR(devices.fbValve_DosingSupply^);
Step5.Command := E_DeviceState.CLOSED;
Step5.StepMinDuration := T#0S;
Step5.DelayUntilNextStep := T#0S;
aSequenceSteps[5] := Step5;
 
Step6.Device := ADR(devices.fbPump_MainPumpA^);
Step6.Command := E_DeviceState.RUNNING;
Step6.StepMinDuration := T#0S;
Step6.DelayUntilNextStep := T#0S;
aSequenceSteps[6] := Step6;
 
Step7.Device := ADR(devices.fbPump_MainPumpB^);
Step7.Command := E_DeviceState.RUNNING;
Step7.StepMinDuration := T#0S;
Step7.DelayUntilNextStep := T#0S;
aSequenceSteps[7] := Step7;
 
Step8.Device := ADR(devices.fbValve_IrrigatorSupply^);
Step8.Command := E_DeviceState.OPEN;
Step8.StepMinDuration := T#0S;
Step8.DelayUntilNextStep := T#0S;
aSequenceSteps[8] := Step8;

nNumberSequenceSteps := 8;  // use this number to limit the number of operations
updateVarIDs();
END_METHOD

END_FUNCTION_BLOCK

// ---- POUs/05 Sequences/Dosing Machine/FB_SequenceDM_Drain.TcPOU
FUNCTION_BLOCK FB_SequenceDM_Drain EXTENDS FB_SequenceBase

VAR
	bUseMainPump_A: BOOL := TRUE;  // this boolean is used to keep track of which of the two redudant pumps we should use
END_VAR

VAR_IN_OUT
	devices: ST_DMComponents;
END_VAR

METHOD FB_init : BOOL
VAR_INPUT
	bInitRetains : BOOL; // if TRUE, the retain variables are initialized (warm start / cold start)
	bInCopyCode : BOOL;  // if TRUE, the instance afterwards gets moved into the copy code (online change)
	
	
END_VAR
(*
		Here we set the order of things to command, what the commands should be, and also how much time to allow during and between steps
		Every component listed below becomes 'Enabled' at each step
*)
sSequenceName := 'DM Drain SEQ';
sSequenceName := 'Dosing Machine Drain sequence';
END_METHOD

METHOD populateSteps : ST_SequenceStep
VAR_INPUT
	
END_VAR
(*
		Here we set the order of things to command, what the commands should be, and also how much time to allow during and between steps
		Every component listed below becomes 'Enabled' at each step
*)
Step1.Device := devices.fbStrainer;
Step1.Command := E_DeviceState.RUNNING;
Step1.StepMinDuration := T#0S; 
Step1.DelayUntilNextStep := T#0S;
aSequenceSteps[1] := Step1;

Step2.Device := devices.fbUnit_UltraSonCleaner;
Step2.Command := E_DeviceState.RUNNING;
Step2.StepMinDuration := T#0S; 
Step2.DelayUntilNextStep := T#0S;
aSequenceSteps[2] := Step2;

Step3.Device := devices.fbUVFilter1;
Step3.Command := E_DeviceState.RUNNING;
Step3.StepMinDuration := T#0S; 
Step3.DelayUntilNextStep := T#10S;				// Steps 1 - 3 can happen in parallel
aSequenceSteps[3] := Step3;

Step4.Device := devices.fbValve_DosingSupply;
Step4.Command := E_DeviceState.OPEN;
Step4.StepMinDuration := T#0S; 
Step4.DelayUntilNextStep := T#0S;
aSequenceSteps[4] := Step4;

(*
Step4.Device := devices.fbPump_MainPumpA;   // start with Pump A - this will need to be changed to pump b every 24hrs
Step1.sID := devices.^.getID();
Step1.sDescr := devices.^.getDescription();
Step4.Command := E_DeviceState.RUNNING;
Step4.StepMinDuration := T#10S; 
Step4.DelayUntilNextStep := T#5S;
aSequenceSteps[4] := Step4;
*)

Step5.Device := devices.fbUnit_OxyInjector;
Step5.Command := E_DeviceState.RUNNING;
Step5.StepMinDuration := T#0S; 
Step5.DelayUntilNextStep := T#0S;
aSequenceSteps[5] := Step5;

Step6.Device := devices.fbDosingPump_phUp;
Step6.Command := E_DeviceState.IDLE;
Step6.StepMinDuration := T#0S; 
Step6.DelayUntilNextStep := T#0S;
aSequenceSteps[6] := Step6;

Step7.Device := devices.fbDosingPump_phDown;
Step7.Command := E_DeviceState.IDLE;
Step7.StepMinDuration := T#0S; 
Step7.DelayUntilNextStep := T#0S;
aSequenceSteps[7] := Step7;

Step8.Device := devices.fbDosingPump_NutrientA;
Step8.Command := E_DeviceState.IDLE;
Step8.StepMinDuration := T#0S; 
Step8.DelayUntilNextStep := T#0S;
aSequenceSteps[8] := Step8;

Step9.Device := devices.fbDosingPump_NutrientB;
Step9.Command := E_DeviceState.IDLE;
Step9.StepMinDuration := T#0S; 
Step9.DelayUntilNextStep := T#0S;
aSequenceSteps[9] := Step9;

Step10.Device := devices.fbDosingPump_NutrientC;
Step10.Command := E_DeviceState.IDLE;
Step10.StepMinDuration := T#0S; 
Step10.DelayUntilNextStep := T#0S;
aSequenceSteps[10] := Step10;



Step11.Device := devices.fbDosingPump_NutrientC;
Step11.Command := E_DeviceState.IDLE;
Step11.StepMinDuration := T#0S; 
Step11.DelayUntilNextStep := T#0S;
aSequenceSteps[11] := Step11;
(* Step11.Component := devices.fbControlLoop_Dosing;
Step11.sID := devices.fbControlLoop_Dosing^.getID();
Step11.sDescr := devices.fbControlLoop_Dosing^.getDescription();
Step11.Command := E_DeviceState.RUNNING;
Step11.StepMinDuration := T#0S; 
Step11.DelayUntilNextStep := T#0S;
aSequenceSteps[11] := Step11;
*)

Step12.Device := devices.fbValve_IrrigatorSupply;
Step12.Command := E_DeviceState.CLOSED;					// This valve may already be closed, sending this command will enable the valve, permitting supervisory control
Step12.StepMinDuration := T#0S; 
Step12.DelayUntilNextStep := T#0S;
aSequenceSteps[12] := Step12;

nNumberSequenceSteps := 12;  // use this number to limit the number of operations
updateVarIDs();
END_METHOD

END_FUNCTION_BLOCK

// ---- POUs/05 Sequences/Dosing Machine/FB_SequenceDM_Fill.TcPOU
FUNCTION_BLOCK FB_SequenceDM_Fill EXTENDS FB_SequenceBase

VAR
	bUseMainPump_A: BOOL := TRUE;  // this boolean is used to keep track of which of the two redudant pumps we should use
END_VAR

VAR_IN_OUT
	devices: ST_DMComponents;
END_VAR

METHOD FB_init : BOOL
VAR_INPUT
	bInitRetains : BOOL; // if TRUE, the retain variables are initialized (warm start / cold start)
	bInCopyCode : BOOL;  // if TRUE, the instance afterwards gets moved into the copy code (online change)
	
	
END_VAR
(*
		Here we set the order of things to command, what the commands should be, and also how much time to allow during and between steps
		Every component listed below becomes 'Enabled' at each step
*)

sSequenceName := 'DM Fill SEQ';
sSequenceName := 'Dosing Machine Fill sequence';
END_METHOD

METHOD populateSteps : ST_SequenceStep
VAR_INPUT
	
END_VAR
(*
		Here we set the order of things to command, what the commands should be, and also how much time to allow during and between steps
		Every component listed below becomes 'Enabled' at each step
*)

Step1.Device := devices.fbStrainer;
Step1.Command := E_DeviceState.RUNNING;
Step1.StepMinDuration := T#0S;
Step1.DelayUntilNextStep := T#0S;
aSequenceSteps[1] := Step1;
 
Step2.Device := devices.fbUnit_UltraSonCleaner;
Step2.Command := E_DeviceState.ON;
Step2.StepMinDuration := T#0S;
Step2.DelayUntilNextStep := T#0S;
aSequenceSteps[2] := Step2;
 
Step3.Device := devices.fbUVFilter1;
Step3.Command := E_DeviceState.ON;
Step3.StepMinDuration := T#0S;
Step3.DelayUntilNextStep := T#0S;
aSequenceSteps[3] := Step3;

Step4.Device := devices.fbValve_DosingSupply;
Step4.Command := E_DeviceState.OPEN;
Step4.StepMinDuration := T#0S;
Step4.DelayUntilNextStep := T#0S;
aSequenceSteps[4] := Step4; 


Step5.Device := devices.fbPump_MainPumpA;
Step5.Command := E_DeviceState.RUNNING;
Step5.StepMinDuration := T#0S;
Step5.DelayUntilNextStep := T#0S;
aSequenceSteps[5] := Step5;
 
Step6.Device := devices.fbPump_MainPumpB;
Step6.Command := E_DeviceState.RUNNING;
Step6.StepMinDuration := T#0S;
Step6.DelayUntilNextStep := T#0S;
aSequenceSteps[6] := Step6;

Step7.Device := devices.fbPump_MainPumpB;
Step7.Device := devices.fbDosingPump_phDown;
Step7.Command := E_DeviceState.RUNNING;
Step7.StepMinDuration := T#0S;
Step7.DelayUntilNextStep := T#0S;
aSequenceSteps[7] := Step7;
 
Step8.Device := devices.fbUnit_OxyInjector;
Step8.Command := E_DeviceState.ON;
Step8.StepMinDuration := T#0S;
Step8.DelayUntilNextStep := T#0S;
aSequenceSteps[8] := Step8;

nNumberSequenceSteps := 8;  // use this number to limit the number of operations 
updateVarIDs();
END_METHOD

END_FUNCTION_BLOCK

// ---- POUs/05 Sequences/Dosing Machine/FB_SequenceDM_Main.TcPOU
FUNCTION_BLOCK FB_SequenceDM_Main EXTENDS FB_SequenceBase

VAR
	bUseMainPump_A: BOOL := TRUE;  // this boolean is used to keep track of which of the two redudant pumps we should use
END_VAR

VAR_IN_OUT
	devices: ST_DMComponents;
END_VAR

METHOD FB_init : BOOL
VAR_INPUT
	bInitRetains : BOOL; // if TRUE, the retain variables are initialized (warm start / cold start)
	bInCopyCode : BOOL;  // if TRUE, the instance afterwards gets moved into the copy code (online change)
	
	
END_VAR
(*
		Here we set the order of things to command, what the commands should be, and also how much time to allow during and between steps
		Every component listed below becomes 'Enabled' at each step
*)
sSequenceName:= 'DM Main Sequence';
sSequenceDescription := 'Main sequence for dosing machine with pH and Nutrient dosing active';
END_METHOD

METHOD populateSteps : ST_SequenceStep
VAR_INPUT
	
END_VAR
(*
		Here we set the order of things to command, what the commands should be, and also how much time to allow during and between steps
		Every component listed below becomes 'Enabled' at each step
*)

Step1.Device := devices.fbStrainer;
Step1.Command := E_DeviceState.RUNNING;
Step1.StepMinDuration := T#5S; 
Step1.DelayUntilNextStep := T#5S;
Step1.WaitForAction := FALSE;
aSequenceSteps[1] := Step1;

Step2.Device := devices.fbStrainer;
Step2.Command := E_DeviceState.RUNNING;
Step2.StepMinDuration := T#5S; 
Step2.DelayUntilNextStep := T#5S;
Step2.WaitForAction := FALSE;
aSequenceSteps[2] := Step2;

Step3.Device := devices.fbUnit_UltraSonCleaner;
Step3.Command := E_DeviceState.RUNNING;
Step3.StepMinDuration := T#5S; 
Step3.DelayUntilNextStep := T#5S;
Step3.WaitForAction := FALSE;
aSequenceSteps[3] := Step3;

Step4.Device := devices.fbUVFilter1;
Step4.Command := E_DeviceState.RUNNING;
Step4.StepMinDuration := T#5S; 
Step4.DelayUntilNextStep := T#5S;				// Steps 1 - 3 can happen in parallel
Step4.WaitForAction := TRUE;
aSequenceSteps[4] := Step4;

Step5.Device := devices.fbValve_DosingSupply;
Step5.Command := E_DeviceState.OPEN;
Step5.StepMinDuration := T#5S; 
Step5.DelayUntilNextStep := T#5S;
Step5.WaitForAction := TRUE;
aSequenceSteps[5] := Step5;

Step6.Device := devices.fbPump_MainPumpA;   // start with Pump A - this will need to be changed to pump b every 24hrs
Step6.Command := E_DeviceState.RUNNING;
Step6.StepMinDuration := T#5S; 
Step6.DelayUntilNextStep := T#5S;
Step6.WaitForAction := TRUE;
aSequenceSteps[6] := Step6;

Step7.Device := devices.fbUnit_OxyInjector;
Step7.Command := E_DeviceState.RUNNING;
Step7.StepMinDuration := T#5S; 
Step7.DelayUntilNextStep := T#5S;
Step7.WaitForAction := FALSE;
aSequenceSteps[7] := Step7;

Step8.Device := devices.fbDosingPump_phUp;
Step8.Command := E_DeviceState.IDLE;
Step8.StepMinDuration := T#5S; 
Step8.DelayUntilNextStep := T#5S;
Step8.WaitForAction := FALSE;
aSequenceSteps[8] := Step8;

Step9.Device := devices.fbDosingPump_phDown;
Step9.Command := E_DeviceState.IDLE;
Step9.StepMinDuration := T#5S; 
Step9.DelayUntilNextStep := T#5S;
Step9.WaitForAction := FALSE;
aSequenceSteps[9] := Step9;

Step10.Device := devices.fbDosingPump_NutrientA;
Step10.Command := E_DeviceState.IDLE;
Step10.StepMinDuration := T#0S; 
Step10.DelayUntilNextStep := T#0S;
Step10.WaitForAction := FALSE;
aSequenceSteps[10] := Step10;

Step11.Device := devices.fbDosingPump_NutrientB;
Step11.Command := E_DeviceState.IDLE;
Step11.StepMinDuration := T#0S; 
Step11.DelayUntilNextStep := T#0S;
Step11.WaitForAction := FALSE;
aSequenceSteps[11] := Step11;

Step12.Device := devices.fbDosingPump_NutrientC;
Step12.Command := E_DeviceState.IDLE;
Step12.StepMinDuration := T#0S; 
Step12.DelayUntilNextStep := T#0S;
Step12.WaitForAction := FALSE;
aSequenceSteps[12] := Step12;


Step13.Device := devices.fbDosingPump_phDown;
Step13.Command := E_DeviceState.IDLE;
Step13.StepMinDuration := T#0S; 
Step13.DelayUntilNextStep := T#0S;
Step13.WaitForAction := FALSE;
aSequenceSteps[13] := Step13;


Step14.Device := devices.fbValve_IrrigatorSupply;
Step14.Command := E_DeviceState.CLOSED;					// This valve may already be closed, sending this command will enable the valve, permitting supervisory control
Step14.StepMinDuration := T#10S; 
Step14.DelayUntilNextStep := T#0S;
Step14.WaitForAction := FALSE;
aSequenceSteps[14] := Step14;

nNumberSequenceSteps := 14;  // use this number to limit the number of operations 
updateVarIDs();
END_METHOD

END_FUNCTION_BLOCK

// ---- POUs/05 Sequences/FB_SequenceManager_ss.TcPOU
(*
		The sequence manager co-ordinates the selection and execution of 
		machine sequences. Machine sequences are created by extending the 
		FB_SequenceBase FB.
*)
FUNCTION_BLOCK FB_SequenceManager_ss
VAR	
	//aSequences: ARRAY[1..5] OF POINTER TO FB_SequenceBase;
	 
	nNumberSequences: INT := 0;
	
	{attribute 'OPC.UA.DA' := '1'} 
	eState:  E_SequenceState := E_SequenceState.STOP; //always stop sequences after PLC restart
	{attribute 'OPC.UA.DA' := '1'} 
	eStateTarget:  E_SequenceState := E_SequenceState.STOP;
	
	eSMState: (STOPPED, STARTING, RUNNING, HOLD) := STOPPED;
	nCurrentStep: INT := 1;
	nCurrentStepPreviousCycle: INT := 1;
	nCurrentSequence: INT := 1;
	nCurrentStepCheck: INT := 1; // use this to iterate over the sequence steps to check if an interlock has rolled back the sequence
	bPauseAcknowledged: BOOL := FALSE;
	
	
	
	{attribute 'OPC.UA.DA' := '0'} 
	fbTONstep: TON;			// these timers are set using the time values stored in each ST_SequenceStep
	{attribute 'OPC.UA.DA' := '0'} 
	fbTONdelay: TON;
	{attribute 'OPC.UA.DA' := '0'} 
	bIsFirstRun: BOOL := TRUE;
	
	i: INT;
	Steps : ARRAY[1..20] OF ST_SequenceStep;
	
	fbCurrentSequence: FB_SequenceBase;
END_VAR

VAR_IN_OUT
	aSequences: ARRAY[1..10] OF FB_SequenceBase;
	//fbCurrentSequence: FB_SequenceBase;
END_VAR

IF bIsFirstRun THEN
	fbTONdelay.PT := T#0S;
	fbTONdelay.IN := TRUE;
	fbTONdelay.PT := T#0S;
	fbTONstep.IN := FALSE;
	bIsFirstRun := FALSE;
	fbCurrentSequence := aSequences[1];
	eSMState := STOPPED;
END_IF


fbTONstep();
fbTONdelay();


CASE eSMState OF
	
	STOPPED:
		// Wait here until a start sequence command is received
		eState := E_SequenceState.STOP;
		
		
	STARTING:
		FOR i := 1 TO fbCurrentSequence.stepsTotal() BY 1 DO
			Steps := fbCurrentSequence.steps();
			Steps[i].Device^.enable();
		END_FOR
	
		nCurrentStepPreviousCycle := nCurrentStep;
		
		// Attempt next step execution 
		IF executeStep(fbCurrentSequence.step(nCurrentStep)) AND nCurrentStep <> fbCurrentSequence.stepsTotal() THEN
			nCurrentStep := nCurrentStep + 1;
		END_IF
		
		
		// Check which sequence step we are up to, set the currentStep indicator to +1 of where we are
		// Interlocks / permissives can cause us to go backwards in steps, therefore we must do this check
		checkCurrentStep();	
		
		IF nCurrentStep < nCurrentStepPreviousCycle THEN  // an interlock has caused the program to roll back in sequence (interlock etc.) - stay in PAUSE state and wait for user acknowledgement
			eSMState := HOLD;
		END_IF
		
			
		IF nCurrentStep = fbCurrentSequence.stepsTotal() THEN  // check if we have completed all of the steps
			eSMState := RUNNING;
		END_IF
		
		eState := E_SequenceState.STARTING;
	
		
		
		
	RUNNING:
		// Sequence is running - just need to check that we are still running, if not, we go to paused
		nCurrentStepPreviousCycle := nCurrentStep;
		checkCurrentStep();
		
		IF nCurrentStep < fbCurrentSequence.stepsTotal() THEN  // something has forced us out of the running state, go to paused and wait for operator to acknowledge
			eSMState := HOLD;
		END_IF
		
		eState := E_SequenceState.RUN;
		
		IF NOT (fbCurrentSequence.step(StepNum := nCurrentStep)^.Device^.getState() = fbCurrentSequence.stepCommand(StepNumber := nCurrentStep)) THEN
			eSMState := STARTING;
		END_IF
		
	HOLD:
		// Do not progress the sequence until the operator has acknowledged that something went wrong
		IF bPauseAcknowledged THEN
			eSMState := STARTING;
			bPauseAcknowledged := FALSE;
		END_IF
		
		eState := E_SequenceState.HOLD;
END_CASE

METHOD acknowledgePause : BOOL
VAR_INPUT
END_VAR
bPauseAcknowledged := TRUE;
END_METHOD

METHOD addSequence : BOOL
VAR_INPUT
	Sequence: FB_SequenceBase;
END_VAR
aSequences[nNumberSequences + 1] := Sequence;
nNumberSequences := nNumberSequences + 1;
END_METHOD

METHOD checkCurrentStep : BOOL
VAR_INPUT
END_VAR

VAR
	currentState: E_DeviceState;
	targetState: E_DeviceState;
END_VAR
nCurrentStepCheck := 1;

WHILE nCurrentStepCheck < (fbCurrentSequence.stepsTotal() + 1) DO
	
	currentState := fbCurrentSequence.stepState(nCurrentStepCheck);
	targetState := fbCurrentSequence.stepCommand(nCurrentStepCheck);

	IF currentState = targetState THEN
		nCurrentStepCheck := nCurrentStepCheck + 1;
	ELSE
		nCurrentStep := nCurrentStepCheck; // step check reveals we are here
		nCurrentStepCheck := fbCurrentSequence.stepsTotal() + 1; // terminate loop as the checking is finished
	END_IF
END_WHILE
END_METHOD

METHOD executeStep : BOOL
VAR_INPUT
	stSequenceStep: POINTER TO ST_SequenceStep;
END_VAR

VAR
	(*eCheckState: E_DeviceState;
	eCheckStateAlternative: E_DeviceState;
	eCheckStateAlternative2: E_DeviceState;
	eCheckCommand: E_DeviceState;
	fbDevice: POINTER TO FB_BaseDevice;
	*)
END_VAR
executeStep := FALSE;
	
// IF fbCurrentSequence.step(StepNum := nCurrentStep)^.Device^.isEnabled()  THEN 
IF (fbCurrentSequence.step(StepNum := nCurrentStep)^.Device^.isEnabled() ) AND 
		(NOT (fbCurrentSequence.step(StepNum := nCurrentStep)^.Device^.getMode() = E_DeviceMode.MANUAL)) THEN 
	//AND fbTONdelay.Q THEN
		
		//fbTONdelay.IN := FALSE; 		
		fbTONstep(IN:= TRUE, PT := stSequenceStep^.StepMinDuration);		
		stSequenceStep^.Device^.setCommand(StateTarget := stSequenceStep^.Command); // set the target state 

END_IF

(*
IF fbCurrentSequence.step(StepNum := nCurrentStep)^.Device^.getState()  
	= fbCurrentSequence.step(StepNum := nCurrentStep)^.Device^.getCommand() 
	AND fbTONstep.Q THEN  *)


IF fbCurrentSequence.step(StepNum := nCurrentStep)^.Device^.getState()  
	= fbCurrentSequence.stepCommand(StepNumber := nCurrentStep)
	AND fbTONstep.Q THEN  
	
	fbTONstep.IN := FALSE; 
	fbTONdelay.IN := FALSE;
	fbTONdelay(IN:= TRUE, PT := stSequenceStep^.DelayUntilNextStep); 
	
	executeStep := TRUE; // indicate that the step was sucessful
	
END_IF
END_METHOD

METHOD getCurrentSeq_FB : POINTER TO FB_SequenceBase
VAR_INPUT
END_VAR
getCurrentSeq_FB := ADR(fbCurrentSequence);
END_METHOD

METHOD getCurrentSeq_ID : INT
VAR_INPUT
END_VAR
getCurrentSeq_ID := nCurrentSequence;
END_METHOD

METHOD getState : E_SequenceState
VAR_INPUT
END_VAR
getState := eState;
END_METHOD

METHOD initSequence : BOOL
VAR_INPUT
END_VAR
// We want to iterate through all of the components in a sequence and enable them.
// We also want to disable any other device (provided it is not in manual)
END_METHOD

METHOD pauseSequence : BOOL
VAR_INPUT
END_VAR
eSMState := HOLD;
END_METHOD

METHOD selectSequence : BOOL
VAR_INPUT
	Sequence: INT;
END_VAR
fbCurrentSequence := aSequences[Sequence];
nCurrentSequence := Sequence;
END_METHOD

METHOD startSequence : BOOL
VAR_INPUT
END_VAR
VAR

END_VAR
eSMState := STARTING;

FOR i := 1 TO fbCurrentSequence.stepsTotal() BY 1 DO
	Steps := fbCurrentSequence.steps();
	Steps[i].Device^.enable();
END_FOR

nCurrentStep := 1;
nCurrentStepPreviousCycle := 1;
//nCurrentSequence := 1;
nCurrentStepCheck := 1;
END_METHOD

METHOD stopSequence : BOOL
VAR_INPUT
END_VAR
eSMState := STOPPED;


FOR i := 1 TO fbCurrentSequence.stepsTotal() BY 1 DO
	Steps := fbCurrentSequence.steps();
	Steps[i].Device^.disable();
END_FOR
END_METHOD

END_FUNCTION_BLOCK

// ---- POUs/05 Sequences/POP/FB_SequenceCONVEY_EXTEND.TcPOU
FUNCTION_BLOCK FB_SequenceCONVEY_EXTEND EXTENDS FB_SequenceBase



VAR_IN_OUT
	devices: ST_POPComponents;
END_VAR

METHOD FB_init : BOOL
VAR_INPUT
	bInitRetains : BOOL; // if TRUE, the retain variables are initialized (warm start / cold start)
	bInCopyCode : BOOL;  // if TRUE, the instance afterwards gets moved into the copy code (online change)
	
	
END_VAR
(*
		Here we set the order of things to command, what the commands should be, and also how much time to allow during and between steps
		Every component listed below becomes 'Enabled' at each step
*)
sSequenceName:= 'POP Conveyor Forward Sequence';
sSequenceDescription := 'Performs the full forward series of actions (starting with tray on static conveyors then lowering onto TRT';
bSequentional_1_Flood_0 := TRUE;
END_METHOD

METHOD populateSteps : ST_SequenceStep
VAR_INPUT
	
END_VAR
(*
		Here we set the order of things to command, what the commands should be, and also how much time to allow during and between steps
		Every component listed below becomes 'Enabled' at each step
*)


Step1.Device := devices.fbTrayCentre_POP1;
Step1.Command := E_DeviceState.RETRACTED;
Step1.StepMinDuration := T#0S;
Step1.DelayUntilNextStep := T#0S;
Step1.WaitForAction := FALSE;
aSequenceSteps[1] :=   Step1;

Step2.Device := devices.fbTrayCentre_POP2;
Step2.Command := E_DeviceState.RETRACTED;
Step2.StepMinDuration := T#0S;
Step2.DelayUntilNextStep := T#0S;
Step2.WaitForAction := FALSE;
aSequenceSteps[2] :=   Step2;

Step3.Device := devices.fbTrayCentre_POP3;
Step3.Command := E_DeviceState.RETRACTED;
Step3.StepMinDuration := T#0S;
Step3.DelayUntilNextStep := T#0S;
Step3.WaitForAction := TRUE;
aSequenceSteps[3] :=   Step3;

Step4.Device := devices.fbStaticConv_POP1;
Step4.Command := E_DeviceState.RUNNING;
Step4.StepMinDuration := T#0S;
Step4.DelayUntilNextStep := T#0S;
Step4.WaitForAction := FALSE;
aSequenceSteps[4] :=   Step4;


Step5.Device := devices.fbStaticConv_POP2;
Step5.Command := E_DeviceState.RUNNING;
Step5.StepMinDuration := T#0S;
Step5.DelayUntilNextStep := T#0S;
Step5.WaitForAction := FALSE;
aSequenceSteps[5] :=   Step5;

Step6.Device := devices.fbStaticConv_POP3;
Step6.Command := E_DeviceState.RUNNING;
Step6.StepMinDuration := T#0S;
Step6.DelayUntilNextStep := T#0S;
Step6.WaitForAction := FALSE;
aSequenceSteps[6] :=   Step9;

Step10.Device := devices.fbTrayEndSensor;
Step10.Command := E_DeviceState.ON;
Step10.StepMinDuration := T#0S;
Step10.DelayUntilNextStep := T#0S;
Step10.WaitForAction := TRUE;
aSequenceSteps[10] :=   Step10;



Step11.Device := devices.fbLinAct_POP1;
Step11.Command := E_DeviceState.RETRACTED;
Step11.StepMinDuration := T#0S; 
Step11.DelayUntilNextStep := T#0S;
Step11.WaitForAction := FALSE;
aSequenceSteps[11] :=   Step11;

Step12.Device := devices.fbLinAct_POP2;
Step12.Command := E_DeviceState.RETRACTED;
Step12.StepMinDuration := T#0S; 
Step12.DelayUntilNextStep := T#0S;
Step12.WaitForAction := FALSE;
aSequenceSteps[12] :=   Step12;

Step13.Device := devices.fbLinAct_POP3;
Step13.Command := E_DeviceState.RETRACTED;
Step13.StepMinDuration := T#0S; 
Step13.DelayUntilNextStep := T#0S;
Step13.WaitForAction := FALSE;
aSequenceSteps[13] :=   Step13;


Step14.Device := devices.fbTrayEndSensor;
Step14.Command := E_DeviceState.OFF;
Step14.StepMinDuration := T#0S; 
Step14.DelayUntilNextStep := T#0S;
Step14.WaitForAction := TRUE;
aSequenceSteps[14] :=   Step14;


nNumberSequenceSteps := 14;  // use this number to limit the number of operations
updateVarIDs();
END_METHOD

END_FUNCTION_BLOCK

// ---- POUs/05 Sequences/POP/FB_SequenceCONVEY_RETRACT.TcPOU
FUNCTION_BLOCK FB_SequenceCONVEY_RETRACT EXTENDS FB_SequenceBase



VAR_IN_OUT
	devices: ST_POPComponents;
END_VAR

METHOD FB_init : BOOL
VAR_INPUT
	bInitRetains : BOOL; // if TRUE, the retain variables are initialized (warm start / cold start)
	bInCopyCode : BOOL;  // if TRUE, the instance afterwards gets moved into the copy code (online change)
	
	
END_VAR
(*
		Here we set the order of things to command, what the commands should be, and also how much time to allow during and between steps
		Every component listed below becomes 'Enabled' at each step
*)
sSequenceName:= 'POP Conveyor Reverse Sequence';
sSequenceDescription := 'Performs the full reverse series of actions (starting with lifting movement and followed by static conveyors';
bSequentional_1_Flood_0 := TRUE;
END_METHOD

METHOD populateSteps : ST_SequenceStep
VAR_INPUT
	
END_VAR
(*
		Here we set the order of things to command, what the commands should be, and also how much time to allow during and between steps
		Every component listed below becomes 'Enabled' at each step
*)

Step1.Device := devices.fbLinAct_POP1;
Step1.Command := E_DeviceState.RETRACTED;
Step1.StepMinDuration := T#0S; 
Step1.DelayUntilNextStep := T#0S;
Step1.WaitForAction := FALSE;
aSequenceSteps[1] :=   Step1;

Step2.Device := devices.fbLinAct_POP1;
Step2.Command := E_DeviceState.RETRACTED;
Step2.StepMinDuration := T#0S; 
Step2.DelayUntilNextStep := T#0S;
Step2.WaitForAction := FALSE;
aSequenceSteps[2] :=   Step2;

Step3.Device := devices.fbLinAct_POP2;
Step3.Command := E_DeviceState.RETRACTED;
Step3.StepMinDuration := T#0S;
Step3.DelayUntilNextStep := T#0S;
Step3.WaitForAction := FALSE;
aSequenceSteps[3] :=   Step3;

Step4.Device := devices.fbTrayCentre_POP1;
Step4.Command := E_DeviceState.RETRACTED;
Step4.StepMinDuration := T#0S;
Step4.DelayUntilNextStep := T#0S;
Step4.WaitForAction := FALSE;
aSequenceSteps[4] :=   Step4;

Step5.Device := devices.fbTrayCentre_POP2;
Step5.Command := E_DeviceState.RETRACTED;
Step5.StepMinDuration := T#0S;
Step5.DelayUntilNextStep := T#0S;
Step5.WaitForAction := FALSE;
aSequenceSteps[5] :=   Step5;

Step6.Device := devices.fbTrayCentre_POP3;
Step6.Command := E_DeviceState.RETRACTED;
Step6.StepMinDuration := T#0S;
Step6.DelayUntilNextStep := T#0S;
Step6.WaitForAction := FALSE;
aSequenceSteps[6] :=   Step6;

Step7.Device := devices.fbTrayEndSensor;
Step7.Command := E_DeviceState.ON;
Step7.StepMinDuration := T#0S;
Step7.DelayUntilNextStep := T#0S;
Step7.WaitForAction := TRUE;
aSequenceSteps[6] :=   Step7;


Step8.Device := devices.fbLinAct_POP1;
Step8.Command := E_DeviceState.EXTENDED;
Step8.StepMinDuration := T#0S;
Step8.DelayUntilNextStep := T#0S;
Step8.WaitForAction := FALSE;
aSequenceSteps[8] :=   Step8;

Step9.Device := devices.fbLinAct_POP2;
Step9.Command := E_DeviceState.EXTENDED;
Step9.StepMinDuration := T#0S;
Step9.DelayUntilNextStep := T#0S;
Step9.WaitForAction := FALSE;
aSequenceSteps[9] :=   Step9;

Step10.Device := devices.fbLinAct_POP3;
Step10.Command := E_DeviceState.EXTENDED;
Step10.StepMinDuration := T#0S;
Step10.DelayUntilNextStep := T#0S;
Step10.WaitForAction := TRUE;
aSequenceSteps[10] :=   Step10;

Step11.Device := devices.fbStaticConv_POP1;
Step11.Command := E_DeviceState.RUNNING;
Step11.StepMinDuration := T#0S; 
Step11.DelayUntilNextStep := T#0S;
Step11.WaitForAction := FALSE;
aSequenceSteps[11] :=   Step11;

Step12.Device := devices.fbStaticConv_POP2;
Step12.Command := E_DeviceState.RUNNING;
Step12.StepMinDuration := T#0S; 
Step12.DelayUntilNextStep := T#0S;
Step12.WaitForAction := FALSE;
aSequenceSteps[12] :=   Step12;

Step13.Device := devices.fbStaticConv_POP3;
Step13.Command := E_DeviceState.RUNNING;
Step13.StepMinDuration := T#0S; 
Step13.DelayUntilNextStep := T#0S;
Step13.WaitForAction := FALSE;
aSequenceSteps[13] :=   Step13;


Step14.Device := devices.fbTrayEndSensor;
Step14.Command := E_DeviceState.OFF;
Step14.StepMinDuration := T#0S; 
Step14.DelayUntilNextStep := T#0S;
Step14.WaitForAction := TRUE;
aSequenceSteps[14] :=   Step14;


nNumberSequenceSteps := 14;  // use this number to limit the number of operations
updateVarIDs();
END_METHOD

END_FUNCTION_BLOCK

// ---- POUs/05 Sequences/POP/FB_SequenceEXTEND_CONVEY.TcPOU
FUNCTION_BLOCK FB_SequenceEXTEND_CONVEY EXTENDS FB_SequenceBase



VAR_IN_OUT
	devices: ST_POPComponents;
END_VAR

METHOD FB_init : BOOL
VAR_INPUT
	bInitRetains : BOOL; // if TRUE, the retain variables are initialized (warm start / cold start)
	bInCopyCode : BOOL;  // if TRUE, the instance afterwards gets moved into the copy code (online change)
	
	
END_VAR
(*
		Here we set the order of things to command, what the commands should be, and also how much time to allow during and between steps
		Every component listed below becomes 'Enabled' at each step
*)
sSequenceName:= 'POP Conveyor Forward Sequence';
sSequenceDescription := 'Performs the full forward series of actions (starting with tray on static conveyors then lowering onto TRT';
bSequentional_1_Flood_0 := TRUE;
END_METHOD

METHOD populateSteps : ST_SequenceStep
VAR_INPUT
	
END_VAR
(*
		Here we set the order of things to command, what the commands should be, and also how much time to allow during and between steps
		Every component listed below becomes 'Enabled' at each step
*)


Step1.Device := devices.fbLinAct_POP1;
Step1.Command := E_DeviceState.RETRACTED;
Step1.StepMinDuration := T#0S; 
Step1.DelayUntilNextStep := T#0S;
Step1.WaitForAction := FALSE;
aSequenceSteps[1] :=   Step1;

Step2.Device := devices.fbLinAct_POP2;
Step2.Command := E_DeviceState.RETRACTED;
Step2.StepMinDuration := T#0S; 
Step2.DelayUntilNextStep := T#0S;
Step2.WaitForAction := FALSE;
aSequenceSteps[2] :=   Step2;

Step3.Device := devices.fbLinAct_POP3;
Step3.Command := E_DeviceState.RETRACTED;
Step3.StepMinDuration := T#0S;
Step3.DelayUntilNextStep := T#0S;
Step3.WaitForAction := FALSE;
aSequenceSteps[3] :=   Step3;

Step4.Device := devices.fbTrayEndSensor;
Step4.Command := E_DeviceState.ON;
Step4.StepMinDuration := T#0S;
Step4.DelayUntilNextStep := T#0S;
Step4.WaitForAction := TRUE;
aSequenceSteps[4] :=   Step4;

Step5.Device := devices.fbTrayCentre_POP1;
Step5.Command := E_DeviceState.RETRACTED;
Step5.StepMinDuration := T#0S;
Step5.DelayUntilNextStep := T#0S;
Step5.WaitForAction := FALSE;
aSequenceSteps[5] :=   Step5;

Step6.Device := devices.fbTrayCentre_POP2;
Step6.Command := E_DeviceState.RETRACTED;
Step6.StepMinDuration := T#0S;
Step6.DelayUntilNextStep := T#0S;
Step6.WaitForAction := FALSE;
aSequenceSteps[6] :=   Step6;

Step7.Device := devices.fbTrayCentre_POP3;
Step7.Command := E_DeviceState.RETRACTED;
Step7.StepMinDuration := T#0S;
Step7.DelayUntilNextStep := T#0S;
Step7.WaitForAction := TRUE;
aSequenceSteps[7] :=   Step7;

Step8.Device := devices.fbStaticConv_POP1;
Step8.Command := E_DeviceState.RUNNING;
Step8.StepMinDuration := T#0S;
Step8.DelayUntilNextStep := T#0S;
Step8.WaitForAction := FALSE;
aSequenceSteps[8] :=   Step8;


Step9.Device := devices.fbStaticConv_POP2;
Step9.Command := E_DeviceState.RUNNING;
Step9.StepMinDuration := T#0S;
Step9.DelayUntilNextStep := T#0S;
Step9.WaitForAction := FALSE;
aSequenceSteps[9] :=   Step9;

Step10.Device := devices.fbStaticConv_POP3;
Step10.Command := E_DeviceState.RUNNING;
Step10.StepMinDuration := T#0S;
Step10.DelayUntilNextStep := T#0S;
Step10.WaitForAction := TRUE;
aSequenceSteps[10] :=   Step10;

Step11.Device := devices.fbTrayEndSensor;
Step11.Command := E_DeviceState.OFF;
Step11.StepMinDuration := T#0S;
Step11.DelayUntilNextStep := T#0S;
Step11.WaitForAction := TRUE;
aSequenceSteps[11] :=   Step11;

Step12.Device := devices.fbLinAct_POP1;
Step12.Command := E_DeviceState.RETRACTED;
Step12.StepMinDuration := T#0S; 
Step12.DelayUntilNextStep := T#0S;
Step12.WaitForAction := FALSE;
aSequenceSteps[12] :=   Step12;

Step13.Device := devices.fbLinAct_POP2;
Step13.Command := E_DeviceState.RETRACTED;
Step13.StepMinDuration := T#0S; 
Step13.DelayUntilNextStep := T#0S;
Step13.WaitForAction := FALSE;
aSequenceSteps[13] :=   Step13;

Step14.Device := devices.fbLinAct_POP3;
Step14.Command := E_DeviceState.RETRACTED;
Step14.StepMinDuration := T#0S; 
Step14.DelayUntilNextStep := T#0S;
Step14.WaitForAction := FALSE;
aSequenceSteps[14] :=   Step14;


Step15.Device := devices.fbTrayEndSensor;
Step15.Command := E_DeviceState.OFF;
Step15.StepMinDuration := T#0S; 
Step15.DelayUntilNextStep := T#0S;
Step15.WaitForAction := TRUE;
aSequenceSteps[15] :=   Step15;


nNumberSequenceSteps := 15;  // use this number to limit the number of operations
updateVarIDs();
END_METHOD

END_FUNCTION_BLOCK

// ---- POUs/05 Sequences/POP/FB_SequenceGET_READY_EXTEND.TcPOU
FUNCTION_BLOCK FB_SequenceGET_READY_EXTEND EXTENDS FB_SequenceBase



VAR_IN_OUT
	devices: ST_POPComponents;
END_VAR

METHOD FB_init : BOOL
VAR_INPUT
	bInitRetains : BOOL; // if TRUE, the retain variables are initialized (warm start / cold start)
	bInCopyCode : BOOL;  // if TRUE, the instance afterwards gets moved into the copy code (online change)
	
	
END_VAR
(*
		Here we set the order of things to command, what the commands should be, and also how much time to allow during and between steps
		Every component listed below becomes 'Enabled' at each step
*)
sSequenceName:= 'POP Conveyor Reverse Sequence';
sSequenceDescription := 'Performs the full reverse series of actions (starting with lifting movement and followed by static conveyors';
bSequentional_1_Flood_0 := TRUE;
END_METHOD

METHOD populateSteps : ST_SequenceStep
VAR_INPUT
	
END_VAR
(*
		Here we set the order of things to command, what the commands should be, and also how much time to allow during and between steps
		Every component listed below becomes 'Enabled' at each step
*)

Step1.Device := devices.fbLinAct_POP1;
Step1.Command := E_DeviceState.EXTENDED;
Step1.StepMinDuration := T#0S; 
Step1.DelayUntilNextStep := T#0S;
Step1.WaitForAction := FALSE;
aSequenceSteps[1] :=   Step1;

Step2.Device := devices.fbLinAct_POP1;
Step2.Command := E_DeviceState.EXTENDED;
Step2.StepMinDuration := T#0S; 
Step2.DelayUntilNextStep := T#0S;
Step2.WaitForAction := FALSE;
aSequenceSteps[2] :=   Step2;

Step3.Device := devices.fbLinAct_POP2;
Step3.Command := E_DeviceState.EXTENDED;
Step3.StepMinDuration := T#0S;
Step3.DelayUntilNextStep := T#0S;
Step3.WaitForAction := FALSE;
aSequenceSteps[3] :=   Step3;

Step4.Device := devices.fbTrayCentre_POP1;
Step4.Command := E_DeviceState.RETRACTED;
Step4.StepMinDuration := T#0S;
Step4.DelayUntilNextStep := T#0S;
Step4.WaitForAction := FALSE;
aSequenceSteps[4] :=   Step4;

Step5.Device := devices.fbTrayCentre_POP2;
Step5.Command := E_DeviceState.RETRACTED;
Step5.StepMinDuration := T#0S;
Step5.DelayUntilNextStep := T#0S;
Step5.WaitForAction := FALSE;
aSequenceSteps[5] :=   Step5;

Step6.Device := devices.fbTrayCentre_POP3;
Step6.Command := E_DeviceState.RETRACTED;
Step6.StepMinDuration := T#0S;
Step6.DelayUntilNextStep := T#0S;
Step6.WaitForAction := FALSE;
aSequenceSteps[6] :=   Step6;

nNumberSequenceSteps := 6;  // use this number to limit the number of operations
updateVarIDs();
END_METHOD

END_FUNCTION_BLOCK

// ---- POUs/05 Sequences/POP/FB_SequenceGET_READY_RETRACT.TcPOU
FUNCTION_BLOCK FB_SequenceGET_READY_RETRACT EXTENDS FB_SequenceBase



VAR_IN_OUT
	devices: ST_POPComponents;
END_VAR

METHOD FB_init : BOOL
VAR_INPUT
	bInitRetains : BOOL; // if TRUE, the retain variables are initialized (warm start / cold start)
	bInCopyCode : BOOL;  // if TRUE, the instance afterwards gets moved into the copy code (online change)
	
	
END_VAR
(*
		Here we set the order of things to command, what the commands should be, and also how much time to allow during and between steps
		Every component listed below becomes 'Enabled' at each step
*)
sSequenceName:= 'POP Conveyor Reverse Sequence';
sSequenceDescription := 'Performs the full reverse series of actions (starting with lifting movement and followed by static conveyors';
bSequentional_1_Flood_0 := TRUE;
END_METHOD

METHOD populateSteps : ST_SequenceStep
VAR_INPUT
	
END_VAR
(*
		Here we set the order of things to command, what the commands should be, and also how much time to allow during and between steps
		Every component listed below becomes 'Enabled' at each step
*)

Step1.Device := devices.fbLinAct_POP1;
Step1.Command := E_DeviceState.RETRACTED;
Step1.StepMinDuration := T#0S; 
Step1.DelayUntilNextStep := T#0S;
Step1.WaitForAction := FALSE;
aSequenceSteps[1] :=   Step1;

Step2.Device := devices.fbLinAct_POP1;
Step2.Command := E_DeviceState.RETRACTED;
Step2.StepMinDuration := T#0S; 
Step2.DelayUntilNextStep := T#0S;
Step2.WaitForAction := FALSE;
aSequenceSteps[2] :=   Step2;

Step3.Device := devices.fbLinAct_POP2;
Step3.Command := E_DeviceState.RETRACTED;
Step3.StepMinDuration := T#0S;
Step3.DelayUntilNextStep := T#0S;
Step3.WaitForAction := FALSE;
aSequenceSteps[3] :=   Step3;

Step4.Device := devices.fbTrayCentre_POP1;
Step4.Command := E_DeviceState.RETRACTED;
Step4.StepMinDuration := T#0S;
Step4.DelayUntilNextStep := T#0S;
Step4.WaitForAction := FALSE;
aSequenceSteps[4] :=   Step4;

Step5.Device := devices.fbTrayCentre_POP2;
Step5.Command := E_DeviceState.RETRACTED;
Step5.StepMinDuration := T#0S;
Step5.DelayUntilNextStep := T#0S;
Step5.WaitForAction := FALSE;
aSequenceSteps[5] :=   Step5;

Step6.Device := devices.fbTrayCentre_POP3;
Step6.Command := E_DeviceState.RETRACTED;
Step6.StepMinDuration := T#0S;
Step6.DelayUntilNextStep := T#0S;
Step6.WaitForAction := FALSE;
aSequenceSteps[6] :=   Step6;

nNumberSequenceSteps := 6;  // use this number to limit the number of operations
updateVarIDs();
END_METHOD

END_FUNCTION_BLOCK

// ---- POUs/05 Sequences/POP/FB_SequenceRETRACT_CONVEY.TcPOU
FUNCTION_BLOCK FB_SequenceRETRACT_CONVEY EXTENDS FB_SequenceBase



VAR_IN_OUT
	devices: ST_POPComponents;
END_VAR

METHOD FB_init : BOOL
VAR_INPUT
	bInitRetains : BOOL; // if TRUE, the retain variables are initialized (warm start / cold start)
	bInCopyCode : BOOL;  // if TRUE, the instance afterwards gets moved into the copy code (online change)
	
	
END_VAR
(*
		Here we set the order of things to command, what the commands should be, and also how much time to allow during and between steps
		Every component listed below becomes 'Enabled' at each step
*)
sSequenceName:= 'POP Conveyor Reverse Sequence';
sSequenceDescription := 'Performs the full reverse series of actions (starting with lifting movement and followed by static conveyors';
bSequentional_1_Flood_0 := TRUE;
END_METHOD

METHOD populateSteps : ST_SequenceStep
VAR_INPUT
	
END_VAR
(*
		Here we set the order of things to command, what the commands should be, and also how much time to allow during and between steps
		Every component listed below becomes 'Enabled' at each step
*)


Step1.Device := devices.fbLinAct_POP1;
Step1.Command := E_DeviceState.RETRACTED;
Step1.StepMinDuration := T#0S; 
Step1.DelayUntilNextStep := T#0S;
Step1.WaitForAction := FALSE;
aSequenceSteps[1] :=   Step1;

Step2.Device := devices.fbLinAct_POP1;
Step2.Command := E_DeviceState.RETRACTED;
Step2.StepMinDuration := T#0S; 
Step2.DelayUntilNextStep := T#0S;
Step2.WaitForAction := FALSE;
aSequenceSteps[2] :=   Step2;

Step3.Device := devices.fbLinAct_POP2;
Step3.Command := E_DeviceState.RETRACTED;
Step3.StepMinDuration := T#0S;
Step3.DelayUntilNextStep := T#0S;
Step3.WaitForAction := FALSE;
aSequenceSteps[3] :=   Step3;

Step4.Device := devices.fbTrayEndSensor;
Step4.Command := E_DeviceState.ON;
Step4.StepMinDuration := T#0S;
Step4.DelayUntilNextStep := T#0S;
Step4.WaitForAction := TRUE;
aSequenceSteps[4] :=   Step4;

Step5.Device := devices.fbTrayCentre_POP1;
Step5.Command := E_DeviceState.EXTENDED;
Step5.StepMinDuration := T#0S;
Step5.DelayUntilNextStep := T#0S;
Step5.WaitForAction := FALSE;
aSequenceSteps[5] :=   Step5;

Step6.Device := devices.fbTrayCentre_POP2;
Step6.Command := E_DeviceState.EXTENDED;
Step6.StepMinDuration := T#0S;
Step6.DelayUntilNextStep := T#0S;
Step6.WaitForAction := FALSE;
aSequenceSteps[6] :=   Step6;

Step7.Device := devices.fbTrayCentre_POP3;
Step7.Command := E_DeviceState.EXTENDED;
Step7.StepMinDuration := T#0S;
Step7.DelayUntilNextStep := T#0S;
Step7.WaitForAction := TRUE;
aSequenceSteps[7] :=   Step7;

Step8.Device := devices.fbStaticConv_POP1;
Step8.Command := E_DeviceState.RUNNING;
Step8.StepMinDuration := T#0S;
Step8.DelayUntilNextStep := T#0S;
Step8.WaitForAction := FALSE;
aSequenceSteps[8] :=   Step8;


Step9.Device := devices.fbStaticConv_POP2;
Step9.Command := E_DeviceState.RUNNING;
Step9.StepMinDuration := T#0S;
Step9.DelayUntilNextStep := T#0S;
Step9.WaitForAction := FALSE;
aSequenceSteps[9] :=   Step9;

Step10.Device := devices.fbStaticConv_POP3;
Step10.Command := E_DeviceState.RUNNING;
Step10.StepMinDuration := T#0S;
Step10.DelayUntilNextStep := T#0S;
Step10.WaitForAction := TRUE;
aSequenceSteps[10] :=   Step10;

Step11.Device := devices.fbTrayEndSensor;
Step11.Command := E_DeviceState.OFF;
Step11.StepMinDuration := T#0S;
Step11.DelayUntilNextStep := T#0S;
Step11.WaitForAction := TRUE;
aSequenceSteps[11] :=   Step11;

Step12.Device := devices.fbLinAct_POP1;
Step12.Command := E_DeviceState.RETRACTED;
Step12.StepMinDuration := T#0S; 
Step12.DelayUntilNextStep := T#0S;
Step12.WaitForAction := FALSE;
aSequenceSteps[12] :=   Step12;

Step13.Device := devices.fbLinAct_POP2;
Step13.Command := E_DeviceState.RETRACTED;
Step13.StepMinDuration := T#0S; 
Step13.DelayUntilNextStep := T#0S;
Step13.WaitForAction := FALSE;
aSequenceSteps[13] :=   Step13;

Step14.Device := devices.fbLinAct_POP3;
Step14.Command := E_DeviceState.RETRACTED;
Step14.StepMinDuration := T#0S; 
Step14.DelayUntilNextStep := T#0S;
Step14.WaitForAction := FALSE;
aSequenceSteps[14] :=   Step14;


Step15.Device := devices.fbTrayEndSensor;
Step15.Command := E_DeviceState.OFF;
Step15.StepMinDuration := T#0S; 
Step15.DelayUntilNextStep := T#0S;
Step15.WaitForAction := TRUE;
aSequenceSteps[15] :=   Step15;


nNumberSequenceSteps := 15;  // use this number to limit the number of operations
updateVarIDs();
END_METHOD

END_FUNCTION_BLOCK

// ---- POUs/05 Sequences/LFT/FB_SequenceMOVE.TcPOU
FUNCTION_BLOCK FB_SequenceMOVE EXTENDS FB_SequenceBase



VAR_IN_OUT
	devices: ST_LFTComponents;
	
	bExt_1_Ret_0_Step2: BOOL;
	bExt_1_Ret_0_Step8: BOOL;
	
END_VAR

METHOD FB_init : BOOL
VAR_INPUT
	bInitRetains : BOOL; // if TRUE, the retain variables are initialized (warm start / cold start)
	bInCopyCode : BOOL;  // if TRUE, the instance afterwards gets moved into the copy code (online change)
	
	
END_VAR
(*
		Here we set the order of things to command, what the commands should be, and also how much time to allow during and between steps
		Every component listed below becomes 'Enabled' at each step
*)
sSequenceName:= 'LFT Move Sequence';
sSequenceDescription := 'Performs a LFT Cycle of picking up a tray and placing a tray';
bSequentional_1_Flood_0 := TRUE;
END_METHOD

METHOD populateSteps : ST_SequenceStep
VAR_INPUT
	
END_VAR
(*
		Here we set the order of things to command, what the commands should be, and also how much time to allow during and between steps
		Every component listed below becomes 'Enabled' at each step
*)

Step1.Device := devices.fbServo_LiftArm;
Step1.Command := E_DeviceState.RETRACTED;
Step1.StepMinDuration := T#0S;
Step1.DelayUntilNextStep := T#0S;
Step1.WaitForAction := FALSE;
aSequenceSteps[1] :=   Step1;

IF bExt_1_Ret_0_Step2 THEN
	Step2.Command := E_DeviceState.EXTENDED;
ELSE
	Step2.Command := E_DeviceState.RETRACTED;
END_IF

Step2.Device := devices.fbServo_Lift;
Step2.StepMinDuration := T#0S;
Step2.DelayUntilNextStep := T#0S;
Step2.WaitForAction := FALSE;
aSequenceSteps[2] :=   Step2;


Step3.Device := devices.fbServo_LiftArm;
Step3.Command := E_DeviceState.EXTENDED;
Step3.StepMinDuration := T#0S;
Step3.DelayUntilNextStep := T#0S;
Step3.WaitForAction := TRUE;
aSequenceSteps[3] :=   Step3;

Step4.Device := devices.fbValve_Vacuum;
Step4.Command := E_DeviceState.OPEN;
Step4.StepMinDuration := T#0S;
Step4.DelayUntilNextStep := T#0S;
Step4.WaitForAction := FALSE;
aSequenceSteps[4] :=   Step4;


Step5.Device := devices.fbSensor_LiftArmVacuum;
Step5.Command := E_DeviceState.ON;
Step5.StepMinDuration := T#0S;
Step5.DelayUntilNextStep := T#0S;
Step5.WaitForAction := TRUE;
aSequenceSteps[5] :=   Step5;

Step6.Device := devices.fbServo_Lift;
Step6.Command := E_DeviceState.EXTENDED;
Step6.StepMinDuration := T#0S;
Step6.DelayUntilNextStep := T#0S;
Step6.WaitForAction := FALSE;
aSequenceSteps[6] :=   Step6;


Step7.Device := devices.fbServo_LiftArm;
Step7.Command := E_DeviceState.RETRACTED;
Step7.StepMinDuration := T#0S;
Step7.DelayUntilNextStep := T#0S;
Step7.WaitForAction := TRUE;
aSequenceSteps[7] :=   Step7;


IF bExt_1_Ret_0_Step8 THEN
	Step8.Command := E_DeviceState.EXTENDED;
ELSE
	Step8.Command := E_DeviceState.RETRACTED;
END_IF

Step8.Device := devices.fbServo_Lift;
Step8.StepMinDuration := T#0S; 
Step8.DelayUntilNextStep := T#0S;
Step8.WaitForAction := FALSE;
aSequenceSteps[8] :=   Step8;

Step9.Device := devices.fbServo_LiftArm;
Step9.Command := E_DeviceState.EXTENDED;
Step9.StepMinDuration := T#0S; 
Step9.DelayUntilNextStep := T#0S;
Step9.WaitForAction := FALSE;
aSequenceSteps[9] :=   Step9;

Step10.Device := devices.fbValve_Vacuum;
Step10.Command := E_DeviceState.RETRACTED;
Step10.StepMinDuration := T#0S; 
Step10.DelayUntilNextStep := T#0S;
Step10.WaitForAction := FALSE;
aSequenceSteps[10] :=   Step10;


Step11.Device := devices.fbSensor_LiftArmVacuum;
Step11.Command := E_DeviceState.OFF;
Step11.StepMinDuration := T#0S; 
Step11.DelayUntilNextStep := T#0S;
Step11.WaitForAction := TRUE;
aSequenceSteps[11] :=   Step11;


nNumberSequenceSteps := 14;  // use this number to limit the number of operations
updateVarIDs();
END_METHOD

END_FUNCTION_BLOCK

// ---- POUs/05 Sequences/RnD Machines/FB_SequenceRNDWTR_Main.TcPOU
FUNCTION_BLOCK FB_SequenceRNDWTR_Main EXTENDS FB_SequenceBase

VAR
	bUseMainPump_A: BOOL := TRUE;  // this boolean is used to keep track of which of the two redudant pumps we should use
END_VAR

VAR_IN_OUT
	devices: ST_RNDWTRComponents;
END_VAR

METHOD FB_init : BOOL
VAR_INPUT
	bInitRetains : BOOL; // if TRUE, the retain variables are initialized (warm start / cold start)
	bInCopyCode : BOOL;  // if TRUE, the instance afterwards gets moved into the copy code (online change)
	
	
END_VAR
(*
		Here we set the order of things to command, what the commands should be, and also how much time to allow during and between steps
		Every component listed below becomes 'Enabled' at each step
*)
sSequenceName:= 'R&D Rooms Lab WTR Main Sequence';
sSequenceDescription := 'Main sequence for R&D water treatment system';
END_METHOD

METHOD populateSteps : ST_SequenceStep
VAR_INPUT
	
END_VAR
(*
		Here we set the order of things to command, what the commands should be, and also how much time to allow during and between steps
		Every component listed below becomes 'Enabled' at each step
*)
Step1.Device := devices.fbUnit_RO_EDI;
Step1.Command := E_DeviceState.ON;
Step1.StepMinDuration := T#0S; 
Step1.DelayUntilNextStep := T#0S;
Step1.WaitForAction := FALSE;
aSequenceSteps[1] :=   Step1;

(*
Step2.Device := devices.fbUnit_RO_EDI;
Step2.Command := E_DeviceState.ON;
Step2.StepMinDuration := T#0S; 
Step2.DelayUntilNextStep := T#0S;
Step2.WaitForAction := FALSE;
aSequenceSteps[2] :=   Step2;
*)


nNumberSequenceSteps := 1;  // use this number to limit the number of operations
updateVarIDs();

(*

				Step8.Component := devices.
				Step8.Command := E_DeviceState.
				Step8.StepMinDuration := T#5S; 
				Step8.DelayUntilNextStep := T#5S;
				Step8.WaitForAction := TRUE;
				aSequenceSteps[8] :=   Step8;
				
				
				Step9.Component := devices.
				Step9.Command := E_DeviceState.
				Step9.StepMinDuration := T#5S; 
				Step9.DelayUntilNextStep := T#5S;
				Step9.WaitForAction := TRUE;
				aSequenceSteps[9] :=   Step9;
				
				
				Step10.Component := devices.
				Step10.Command := E_DeviceState.
				Step10.StepMinDuration := T#5S; 
				Step10.DelayUntilNextStep := T#5S;
				Step10.WaitForAction := TRUE;
				aSequenceSteps[10] :=   Step10;
				
				
				Step11.Component := devices.
				Step11.Command := E_DeviceState.
				Step11.StepMinDuration := T#5S; 
				Step11.DelayUntilNextStep := T#5S;
				Step11.WaitForAction := TRUE;
				aSequenceSteps[11] :=   Step11;
				
				
				Step12.Component := devices.
				Step12.Command := E_DeviceState.
				Step12.StepMinDuration := T#5S; 
				Step12.DelayUntilNextStep := T#5S;
				Step12.WaitForAction := TRUE;
				aSequenceSteps[12] :=   Step12;
				
				
				Step13.Component := devices.
				Step13.Command := E_DeviceState.
				Step13.StepMinDuration := T#5S; 
				Step13.DelayUntilNextStep := T#5S;
				Step13.WaitForAction := TRUE;
				aSequenceSteps[13] :=   Step13;
				
				
				Step14.Component := devices.
				Step14.Command := E_DeviceState.
				Step14.StepMinDuration := T#5S; 
				Step14.DelayUntilNextStep := T#5S;
				Step14.WaitForAction := TRUE;
				aSequenceSteps[14] :=   Step14;
				
				
				Step15.Component := devices.
				Step15.Command := E_DeviceState.
				Step15.StepMinDuration := T#5S; 
				Step15.DelayUntilNextStep := T#5S;
				Step15.WaitForAction := TRUE;
				aSequenceSteps[15] :=   Step15;
				
				
				Step16.Component := devices.
				Step16.Command := E_DeviceState.
				Step16.StepMinDuration := T#5S; 
				Step16.DelayUntilNextStep := T#5S;
				Step16.WaitForAction := TRUE;
				aSequenceSteps[16] :=   Step16;
				
				
				Step17.Component := devices.
				Step17.Command := E_DeviceState.
				Step17.StepMinDuration := T#5S; 
				Step17.DelayUntilNextStep := T#5S;
				Step17.WaitForAction := TRUE;
				aSequenceSteps[17] :=   Step17;
				
				
				Step18.Component := devices.
				Step18.Command := E_DeviceState.
				Step18.StepMinDuration := T#5S; 
				Step18.DelayUntilNextStep := T#5S;
				Step18.WaitForAction := TRUE;
				aSequenceSteps[18] :=   Step18;
				
				
				Step19.Component := devices.
				Step19.Command := E_DeviceState.
				Step19.StepMinDuration := T#5S; 
				Step19.DelayUntilNextStep := T#5S;
				Step19.WaitForAction := TRUE;
				aSequenceSteps[19] :=   Step19;
				
				
				Step20.Component := devices.
				Step20.Command := E_DeviceState.
				Step20.StepMinDuration := T#5S; 
				Step20.DelayUntilNextStep := T#5S;
				Step20.WaitForAction := TRUE;
				aSequenceSteps[20] :=   Step20;
*)
END_METHOD

END_FUNCTION_BLOCK

// ---- POUs/05 Sequences/RnD Machines/FB_SequenceRND_Calibrate.TcPOU
FUNCTION_BLOCK FB_SequenceRND_Calibrate EXTENDS FB_SequenceBase

VAR
	bUseMainPump_A: BOOL := TRUE;  // this boolean is used to keep track of which of the two redudant pumps we should use
END_VAR

VAR_IN_OUT
	devices: ST_RNDDMComponents;
END_VAR

METHOD FB_init : BOOL
VAR_INPUT
	bInitRetains : BOOL; // if TRUE, the retain variables are initialized (warm start / cold start)
	bInCopyCode : BOOL;  // if TRUE, the instance afterwards gets moved into the copy code (online change)
END_VAR
(*
		Here we set the order of things to command, what the commands should be, and also how much time to allow during and between steps
		Every component listed below becomes 'Enabled' at each step
*)

sSequenceName := 'RND-DM Calibrate SEQ';
sSequenceName := 'R&D Dosing Machine Calibrate sequence';
END_METHOD

METHOD populateSteps : ST_SequenceStep
VAR_INPUT

END_VAR
(*
		Here we set the order of things to command, what the commands should be, and also how much time to allow during and between steps
		Every component listed below becomes 'Enabled' at each step
*)

Step1.Device := devices.fbPump_MainPumpA;
Step1.Command := E_DeviceState.RUNNING;
Step1.StepMinDuration := T#5S; 
Step1.DelayUntilNextStep := T#5S;
Step1.WaitForAction := TRUE;
aSequenceSteps[1] :=   Step1;

Step2.Device := devices.fbUVFilter1;
Step2.Command := E_DeviceState.ON;
Step2.StepMinDuration := T#5S;
Step2.DelayUntilNextStep := T#5S;
Step2.WaitForAction := TRUE;
aSequenceSteps[2] :=   Step2;

Step3.Device := devices.fbControlLoop_TankLevel;
Step3.Command := E_DeviceState.ON;
Step3.DelayUntilNextStep := T#5S;
Step3.StepMinDuration := T#5S;
Step3.DelayUntilNextStep := T#5S;
Step3.WaitForAction := TRUE;
aSequenceSteps[3] :=   Step3;

Step4.Device := devices.fbControlLoop_DissOx;
Step4.Command := E_DeviceState.ON;
Step4.DelayUntilNextStep := T#5S;
Step4.StepMinDuration := T#5S;
Step4.DelayUntilNextStep := T#5S;
Step4.WaitForAction := TRUE;
aSequenceSteps[4] :=   Step4;

Step5.Device := devices.fbControlLoop_Dosing;
Step5.Command := E_DeviceState.ON;
Step5.DelayUntilNextStep := T#5S;
Step5.StepMinDuration := T#5S;
Step5.DelayUntilNextStep := T#5S;
Step5.WaitForAction := TRUE;
aSequenceSteps[5] :=   Step5;

Step6.Device := devices.fbValve_Drain;
Step6.Command := E_DeviceState.CLOSED;
Step6.DelayUntilNextStep := T#5S;
Step6.StepMinDuration := T#5S;
Step6.DelayUntilNextStep := T#5S;
Step6.WaitForAction := TRUE;
aSequenceSteps[6] :=   Step6;


nNumberSequenceSteps := 6;  // use this number to limit the number of operations
updateVarIDs();
END_METHOD

END_FUNCTION_BLOCK

// ---- POUs/05 Sequences/RnD Machines/FB_SequenceRND_Drain.TcPOU
FUNCTION_BLOCK FB_SequenceRND_Drain EXTENDS FB_SequenceBase

VAR
	bUseMainPump_A: BOOL := TRUE;  // this boolean is used to keep track of which of the two redudant pumps we should use
END_VAR

VAR_IN_OUT
	devices: ST_RNDDMComponents;
END_VAR


Step1.Device := devices.fbValve_Drain;
Step1.Command := E_DeviceState.OPEN;
Step1.DelayUntilNextStep := T#5S;
Step1.StepMinDuration := T#5S;
Step1.DelayUntilNextStep := T#5S;
Step1.WaitForAction := TRUE;
aSequenceSteps[1] :=   Step1;

Step2.Device := devices.fbValve_RevOsSupply;
Step2.Command := E_DeviceState.CLOSED;
Step2.DelayUntilNextStep := T#5S;
Step2.StepMinDuration := T#5S;
Step2.DelayUntilNextStep := T#5S;
Step2.WaitForAction := TRUE;
aSequenceSteps[2] :=   Step2;

nNumberSequenceSteps := 2;  // use this number to limit the number of operations
updateVarIDs();

METHOD FB_init : BOOL
VAR_INPUT
	bInitRetains : BOOL; // if TRUE, the retain variables are initialized (warm start / cold start)
	bInCopyCode : BOOL;  // if TRUE, the instance afterwards gets moved into the copy code (online change)
	
	
END_VAR
(*
		Here we set the order of things to command, what the commands should be, and also how much time to allow during and between steps
		Every component listed below becomes 'Enabled' at each step
*)

sSequenceName := 'RND-DM Drain SEQ';
sSequenceName := 'R&D Dosing Machine Drain sequence';
END_METHOD

METHOD populateSteps : ST_SequenceStep
VAR_INPUT
	
END_VAR
(*
		Here we set the order of things to command, what the commands should be, and also how much time to allow during and between steps
		Every component listed below becomes 'Enabled' at each step
*)




Step1.Device := devices.fbValve_RevOsSupply;
Step1.Command := E_DeviceState.CLOSED;
Step1.DelayUntilNextStep := T#5S;
Step1.StepMinDuration := T#5S;
Step1.DelayUntilNextStep := T#5S;
Step1.WaitForAction := TRUE;
aSequenceSteps[1] :=   Step1;


Step2.Device := devices.fbValve_Drain;
Step2.Command := E_DeviceState.OPEN;
Step2.DelayUntilNextStep := T#5S;
Step2.StepMinDuration := T#5S;
Step2.DelayUntilNextStep := T#5S;
Step2.WaitForAction := TRUE;
aSequenceSteps[2] :=   Step2;


nNumberSequenceSteps := 2;  // use this number to limit the number of operations
updateVarIDs();
END_METHOD

END_FUNCTION_BLOCK

// ---- POUs/05 Sequences/RnD Machines/FB_SequenceRND_Fill.TcPOU
FUNCTION_BLOCK FB_SequenceRND_Fill EXTENDS FB_SequenceBase

VAR
	bUseMainPump_A: BOOL := TRUE;  // this boolean is used to keep track of which of the two redudant pumps we should use
END_VAR

VAR_IN_OUT
	devices: ST_RNDDMComponents;
END_VAR

METHOD FB_init : BOOL
VAR_INPUT
	bInitRetains : BOOL; // if TRUE, the retain variables are initialized (warm start / cold start)
	bInCopyCode : BOOL;  // if TRUE, the instance afterwards gets moved into the copy code (online change)
	
	
END_VAR
(*
		Here we set the order of things to command, what the commands should be, and also how much time to allow during and between steps
		Every component listed below becomes 'Enabled' at each step
*)

sSequenceName := 'RND-DM Fill SEQ';
sSequenceName := 'R&D Dosing Machine Fill sequence';
END_METHOD

METHOD populateSteps : ST_SequenceStep
VAR_INPUT
	
